// TwinCAT 3 PLC project Stage
// Title: Stage
// Company: _
// Author: Krystian Lis et al.
// ProjectVersion: 4.1.3
// ProgramVersion: 3.1.4026.22
// libraries:
//   Tc2_Standard, * (Beckhoff Automation GmbH)
//   Tc2_System, * (Beckhoff Automation GmbH)
//   Tc2_Utilities, * (Beckhoff Automation GmbH)
// project tree:
//   Plant/Debugging/ DebugStruct.TcDUT, I_Debug.TcIO
//   Plant/Entity/ Entity.TcPOU, I_Entity.TcIO, _I_Entity.TcIO
//   Plant/Execute/ Execute.TcPOU, I_Execute.TcIO, _I_Execute.TcIO
//   Plant/Init/ I_Init.TcIO
//   Plant/Job/ I_Worker.TcIO, _I_Worker.TcIO, Worker.TcPOU, I_Job.TcIO, JobState.TcDUT
//   Plant/OnlineChange/ I_OnlineChange.TcIO
//   Plant/ Plant.TcPOU, _Plant.TcGVL
//   Plant/PreInit/ I_PreInit.TcIO
//   Plant/PostInit/ I_PostInit.TcIO
//   Plant/Thread/ I_Thread.TcIO, Thread.TcPOU, _I_Thread.TcIO
//   Plant/Validate/ _I_ValidateGeneric.TcIO, I_ValidateInterface.TcIO
//   Utils/Color/ Argb.TcDUT, Argbb.TcPOU, GenArgb.TcPOU
//   Utils/Generic/ I_Generic.TcIO
//   Utils/Math/ Math.TcPOU
//   Utils/Path/ I_Path.TcIO, Path.TcPOU
//   Utils/Result/Error/ GenericResult.TcGVL
//   Utils/Result/ IsErr.TcPOU, IsFail.TcPOU, IsNone.TcPOU, IsOk.TcPOU, IsSome.TcPOU, Result.TcDUT
//   Utils/Strings/Alias/ Ch.TcDUT, Str.TcDUT
//   Utils/Strings/Strb/ I_Strb.TcIO, Strb.TcPOU
//   Utils/Strings/Strf/ Strf.TcPOU
//   Utils/Time/ GetTaskCycleTime.TcPOU, GetUnixTime.TcPOU
//   _/ Param.TcGVL
// real-time tasks:
//   TASK Example: cycle T#10ms, priority 20, ADS port 350
//   TASK Test: cycle T#10ms, priority 21, ADS port 351
//   TASK VISU_TASK: cycle T#200000us, priority 30, ADS port 352
//   TASK PlcTask: cycle T#10ms, priority 22, ADS port 353
//   TASK PlcTask1: cycle T#10ms, priority 23, ADS port 354
//   TASK PlcTask2: cycle T#10ms, priority 24, ADS port 355

// ---- Plant/Debugging/DebugStruct.TcDUT
// One diagnostic entry.
TYPE DebugStruct :
STRUCT
	iSource: I_Debug; // Object that reported the message.
	sComment: Str; // Diagnostic text.
END_STRUCT
END_TYPE

// ---- Plant/Job/JobState.TcDUT
// Worker lifecycle state.
{attribute 'qualified_only'}
{attribute 'strict'}
{attribute 'to_string'}
TYPE JobState :
(
	Idle, // Not attached to a thread.
	Init, // Will call JobInit next.
	Busy, // Calls JobExecute each worker cycle.
	Done // Will call JobExit and detach.
	
) BYTE;
END_TYPE

// ---- Utils/Color/Argb.TcDUT
// Packed ARGB color value.
TYPE Argb : DWORD; END_TYPE

// ---- Utils/Result/Result.TcDUT
// Result code: >0 Ok, 0 None, <0 Error.
TYPE Result : INT; END_TYPE

// ---- Utils/Strings/Alias/Ch.TcDUT
// Single-character string alias.
TYPE Ch : STRING(1); END_TYPE

// ---- Utils/Strings/Alias/Str.TcDUT
// Common 255-character string alias.
TYPE Str : STRING(255); END_TYPE

// ---- Plant/_Plant.TcGVL
{attribute 'qualified_only'}
{attribute 'global_init_slot' := '40001'}
VAR_GLOBAL INTERNAL
	panic: ARRAY[1..PARAM.MAX_PANIC_MSG] OF DebugStruct;
	warn: ARRAY[1..PARAM.MAX_WARN_MSG] OF DebugStruct;
	
	nLastPanic: UDINT := 1;
	nLastWarn: UDINT := 1;
	nTotalPanic: UDINT;
	nTotalWarn: UDINT;
	
	{attribute 'init_on_onlchange'}
	bOnlineChange: BOOL := TRUE;
	
	{attribute 'no_copy'}
	{attribute 'no_init'}
	bOnlineChangeEntityCreated: BOOL := FALSE;
	{attribute 'no_copy'}
	{attribute 'no_init'}
	bOnlineChangeEntityDeleted: BOOL := FALSE;

	iFirstThread: I_Thread;
	iLastThread: I_Thread;

	iFirstWorker: I_Worker;
	iLastWorker: I_Worker;
	
	MainThread: Thread;
	
	iFirstEntity: I_Entity;
	iLastEntity: I_Entity;
	
	bPanic: BOOL;
	bInit: BOOL := TRUE;
END_VAR

// ---- Utils/Result/Error/GenericResult.TcGVL
VAR_GLOBAL CONSTANT
	None	: Result := 0; // No result or end of iteration.
	Ok		: Result := 1; // Generic success.
	Error	: Result := -1; // Generic error.
END_VAR

// ---- _/Param.TcGVL
// Stage diagnostic buffer limits.
{attribute 'qualified_only'}
VAR_GLOBAL CONSTANT
	MAX_PANIC_MSG: UDINT(1..16#7FFFFFFF) := 10; // Panic buffer entries; do not set to 0.
	MAX_WARN_MSG: UDINT(1..16#7FFFFFFF) := 10; // Warning buffer entries; do not set to 0.
	VALIDATION_GUARD: UDINT(1..16#7FFFFFFF) := 100_000;
END_VAR

// ---- Plant/Debugging/I_Debug.TcIO
// Diagnostic marker interface.
INTERFACE I_Debug

END_INTERFACE

// ---- Plant/Entity/I_Entity.TcIO
// Registered entity handle.
INTERFACE I_Entity EXTENDS _I_Entity

// Raw discoverable interface for __QUERYINTERFACE.
PROPERTY Raw : I_Generic
GET
END_GET
END_PROPERTY

END_INTERFACE

// ---- Plant/Entity/_I_Entity.TcIO
INTERFACE INTERNAL _I_Entity EXTENDS I_Debug, I_ValidateInterface

METHOD INTERNAL GetNext : I_Entity
END_METHOD

METHOD INTERNAL SetNext
VAR_INPUT
	iNext: I_Entity;
END_VAR
END_METHOD

METHOD INTERNAL GetPrev : I_Entity
END_METHOD

METHOD INTERNAL SetPrev
VAR_INPUT
	iPrev: I_Entity;
END_VAR
END_METHOD

METHOD INTERNAL GetRaw : I_Generic
END_METHOD

METHOD INTERNAL SetRaw
VAR_INPUT
	iRaw: I_Generic;
END_VAR
END_METHOD

PROPERTY INTERNAL _Result : Result
GET
END_GET
END_PROPERTY

PROPERTY INTERNAL _NewInstance : BOOL
GET
END_GET
SET
END_SET
END_PROPERTY

END_INTERFACE

// ---- Plant/Execute/I_Execute.TcIO
// Cyclic callback contract; Execute is called once per assigned thread cycle.
INTERFACE I_Execute EXTENDS I_Debug

// Called cyclically by the assigned Stage thread.
METHOD Execute
END_METHOD

END_INTERFACE

// ---- Plant/Execute/_I_Execute.TcIO
INTERFACE INTERNAL _I_Execute EXTENDS I_Debug, I_ValidateInterface;

METHOD INTERNAL _Exe
VAR_OUTPUT
	iNext: _I_Execute;
END_VAR
END_METHOD

METHOD INTERNAL GetNext : _I_Execute
END_METHOD

METHOD INTERNAL SetNext
VAR_INPUT
	iNext: _I_Execute;
END_VAR
END_METHOD

METHOD INTERNAL GetPrev : _I_Execute
END_METHOD

METHOD INTERNAL SetPrev
VAR_INPUT
	iPrev: _I_Execute;
END_VAR
END_METHOD

METHOD INTERNAL GetThread : I_Thread
END_METHOD

METHOD INTERNAL SetThread
VAR_INPUT
	iThread: I_Thread;
END_VAR
END_METHOD

END_INTERFACE

// ---- Plant/Init/I_Init.TcIO
// Startup hook called after PreInit and before PostInit.
INTERFACE I_Init EXTENDS I_Generic

// Called once during Plant startup.
METHOD Init
END_METHOD

END_INTERFACE

// ---- Plant/Job/I_Worker.TcIO
// Public command interface for a Worker.
INTERFACE I_Worker EXTENDS _I_Worker

// Starts idle job; returns Ok attached, None command busy, Error invalid state or job.
METHOD Start : Result
VAR_INPUT
END_VAR
END_METHOD

// Current worker state.
PROPERTY State : JobState
GET
END_GET
END_PROPERTY

// Requests stop; Busy moves to Done and calls JobExit before returning Idle.
METHOD Stop
VAR_INPUT
END_VAR
END_METHOD

END_INTERFACE

// ---- Plant/Job/_I_Worker.TcIO
INTERFACE INTERNAL _I_Worker EXTENDS I_Debug, I_ValidateInterface;

METHOD INTERNAL GetNext : I_Worker
END_METHOD

METHOD INTERNAL SetNext
VAR_INPUT
	iNext: I_Worker;
END_VAR
END_METHOD

METHOD INTERNAL GetPrev : I_Worker
END_METHOD

METHOD INTERNAL SetPrev
VAR_INPUT
	iPrev: I_Worker;
END_VAR
END_METHOD

METHOD INTERNAL GetPlantNext : I_Worker
END_METHOD

METHOD INTERNAL SetPlantNext
VAR_INPUT
	iNext: I_Worker;
END_VAR
END_METHOD

METHOD INTERNAL GetPlantPrev : I_Worker
END_METHOD

METHOD INTERNAL SetPlantPrev
VAR_INPUT
	iPrev: I_Worker;
END_VAR
END_METHOD

METHOD INTERNAL Process
VAR_OUTPUT
	iNext: I_Worker;
END_VAR
END_METHOD

METHOD INTERNAL GetThread : I_Thread
END_METHOD

METHOD INTERNAL SetThread
VAR_INPUT
	iThread: I_Thread;
END_VAR
END_METHOD

END_INTERFACE

// ---- Plant/Job/I_Job.TcIO
// Startable job contract processed by Worker.
INTERFACE I_Job EXTENDS I_Debug

// Called every worker cycle while Busy.
METHOD JobExecute
VAR_INPUT
END_VAR
END_METHOD

// Called once when the worker leaves Done.
METHOD JobExit
VAR_INPUT
END_VAR
END_METHOD

// Called once when the worker enters Init.
METHOD JobInit
VAR_INPUT
END_VAR
END_METHOD

END_INTERFACE

// ---- Plant/OnlineChange/I_OnlineChange.TcIO
INTERFACE I_OnlineChange EXTENDS I_Generic

METHOD OnOnlineChange
VAR_INPUT
	bEntityDeleted: BOOL;
	bEntityCreated: BOOL;
END_VAR
END_METHOD

END_INTERFACE

// ---- Plant/PreInit/I_PreInit.TcIO
// Startup hook called before Init and PostInit.
INTERFACE I_PreInit EXTENDS I_Generic

// Called once during Plant startup before Init.
METHOD PreInit
END_METHOD

END_INTERFACE

// ---- Plant/PostInit/I_PostInit.TcIO
// Startup hook called after PreInit and Init.
INTERFACE I_PostInit EXTENDS I_Generic

// Called once during Plant startup after Init.
METHOD PostInit
END_METHOD

END_INTERFACE

// ---- Plant/Thread/I_Thread.TcIO
// Identifies a Stage execution thread.
INTERFACE I_Thread EXTENDS _I_Thread

END_INTERFACE

// ---- Plant/Thread/_I_Thread.TcIO
INTERFACE INTERNAL _I_Thread EXTENDS I_Debug, I_ValidateInterface

METHOD INTERNAL GetFirst : _I_Execute
END_METHOD

METHOD INTERNAL GetFirstWorker : I_Worker
END_METHOD

METHOD INTERNAL GetLast : _I_Execute
END_METHOD

METHOD INTERNAL GetLastWorker : I_Worker
END_METHOD

METHOD INTERNAL GetNext : I_Thread
END_METHOD

METHOD INTERNAL SetNext
VAR_INPUT
	iNext: I_Thread;
END_VAR
END_METHOD

METHOD INTERNAL GetPrev : I_Thread
END_METHOD

METHOD INTERNAL SetPrev
VAR_INPUT
	iPrev: I_Thread;
END_VAR
END_METHOD

METHOD INTERNAL AttachExecute : Result
VAR_INPUT
	iExecute: _I_Execute;
END_VAR
END_METHOD

METHOD INTERNAL AttachWorker : Result
VAR_INPUT
	iWorker: I_Worker;
END_VAR
END_METHOD

METHOD INTERNAL DetachExecute : Result
VAR_INPUT
	iExecute: _I_Execute;
END_VAR
END_METHOD

METHOD INTERNAL DetachWorker : Result
VAR_INPUT
	iWorker: I_Worker;
END_VAR
END_METHOD

METHOD INTERNAL ValidateThread : Result
END_METHOD

END_INTERFACE

// ---- Plant/Validate/_I_ValidateGeneric.TcIO
INTERFACE INTERNAL _I_ValidateGeneric EXTENDS __SYSTEM.IQueryInterface, I_Debug

END_INTERFACE

// ---- Plant/Validate/I_ValidateInterface.TcIO
INTERFACE I_ValidateInterface EXTENDS I_Debug

{attribute 'hide'}
METHOD ValidateInterface
VAR_INPUT
END_VAR
END_METHOD

END_INTERFACE

// ---- Utils/Generic/I_Generic.TcIO
// Common discoverable base interface for registered entities.
INTERFACE I_Generic EXTENDS __SYSTEM.IQueryInterface, I_Debug

END_INTERFACE

// ---- Utils/Path/I_Path.TcIO
// Path identifier interface.
INTERFACE I_Path

// Full generated path including options.
PROPERTY Get : Str
GET
END_GET
END_PROPERTY

// TRUE when the path contains sSegment.
METHOD Has : BOOL
VAR_INPUT
	sSegment: Str; // Segment to find.
END_VAR
END_METHOD

// Full path length including options.
PROPERTY Length : USINT
GET
END_GET
END_PROPERTY

// Generated path without options.
PROPERTY Name : Str
GET
END_GET
END_PROPERTY

// Optional query-style path segment.
PROPERTY Option : Str
GET
END_GET
SET
END_SET
END_PROPERTY

END_INTERFACE

// ---- Utils/Strings/Strb/I_Strb.TcIO
// Chainable string builder interface.
INTERFACE INTERNAL I_Strb EXTENDS I_Debug

// Appends text; truncates at 255 chars.
METHOD Append : I_Strb
VAR_INPUT
    sToAdd : Str; // Text to append.
END_VAR
END_METHOD

// Finds first match after position; outputs zero positions when not found.
METHOD FindFirstAfter : I_Strb
VAR_INPUT
    sToFind : Str;      // Text to find.
    nPosition : INT := 1; // One-based start position.
END_VAR
VAR_OUTPUT
    nStart : INT;       // Match start, or 0.
    nEnd : INT;         // Match end, or 0.
END_VAR
END_METHOD

// Finds last match before position; outputs zero positions when not found.
METHOD FindLastBefore : I_Strb
VAR_INPUT
    sToFind : Str;        // Text to find.
    nPosition : INT := 256; // One-based end position; 256 means current length.
END_VAR
VAR_OUTPUT
    nStart : INT;         // Match start, or 0.
    nEnd : INT;           // Match end, or 0.
END_VAR
END_METHOD

// Returns current text.
METHOD Get : Str
VAR_INPUT
END_VAR
END_METHOD

// Returns current length.
METHOD GetLength : INT
VAR_INPUT
END_VAR
END_METHOD

// TRUE when text is found after position.
METHOD HasAfter : BOOL
VAR_INPUT
    sToFind : Str;      // Text to find.
    nPosition : INT := 0; // One-based start position.
END_VAR
VAR_OUTPUT
    nStart : INT;       // Match start, or 0.
    nEnd : INT;         // Match end, or 0.
END_VAR
END_METHOD

// TRUE when text is found before position.
METHOD HasBefore : BOOL
VAR_INPUT
    sToFind : Str;        // Text to find.
    nPosition : INT := 256; // One-based end position; 256 means current length.
END_VAR
VAR_OUTPUT
    nStart : INT;         // Match start, or 0.
    nEnd : INT;           // Match end, or 0.
END_VAR
END_METHOD

// Inserts text; no change when position is invalid.
METHOD Inject : I_Strb
VAR_INPUT
    nPosition : INT;    // One-based insert position.
    sToInject : Str;    // Text to insert.
END_VAR
END_METHOD

// TRUE when current length is 0.
METHOD IsEmpty : BOOL
VAR_INPUT
END_VAR
END_METHOD

// Outputs current length and returns this builder.
METHOD Length : I_Strb
VAR_OUTPUT
	nLen: INT; // Current length.
END_VAR
END_METHOD

// Prepends text; truncates at 255 chars.
METHOD Prepend : I_Strb
VAR_INPUT
    sToAdd : Str; // Text to prepend.
END_VAR
END_METHOD

// Removes text; no change when position or length is invalid.
METHOD Remove : I_Strb
VAR_INPUT
    nLength : INT;    // Characters to remove.
    nPosition : INT;  // One-based start position.
END_VAR
END_METHOD

// Sets current text.
METHOD Set : I_Strb
VAR_INPUT
    sValue : Str; // New text.
END_VAR
END_METHOD

// Copies substring into sSlice; no change when position or length is invalid.
METHOD Slice : I_Strb
VAR_INPUT
	nLength : INT;   // Characters to copy.
    nPosition : INT; // One-based start position.
END_VAR
VAR_OUTPUT
    sSlice : Strb;   // Output slice builder.
END_VAR
END_METHOD

// Splits text into left and right builders.
METHOD Split : I_Strb
VAR_INPUT
    nPosition : INT; // One-based split position.
END_VAR
VAR_OUTPUT
    sLeft : Strb;    // Left side.
    sRight : Strb;   // Right side.
END_VAR
END_METHOD

// Outputs current text and returns this builder.
METHOD Write : I_Strb;
VAR_OUTPUT
	sOut: Str; // Current text.
END_VAR
END_METHOD

END_INTERFACE

// ---- Plant/Thread/Thread.TcPOU
// Runs executors and active workers assigned to this TwinCAT task.
FUNCTION_BLOCK Thread IMPLEMENTS I_Thread
VAR
	iFirstExecute: _I_Execute;
	iLastExecute: _I_Execute;

	iFirstWorker: I_Worker;
	iLastWorker: I_Worker;

	iPrevThread: I_Thread;
	iNextThread: I_Thread;
END_VAR

METHOD INTERNAL AttachExecute : Result
VAR_INPUT
	iExecute: _I_Execute;
END_VAR
VAR
	iThis: I_Thread := THIS^;
	iThread: I_Thread;
	iPrev: _I_Execute;
	iNext: _I_Execute;
END_VAR
IF iExecute = 0 THEN
	AttachExecute := Error;
	RETURN;
END_IF

iThread := iExecute.GetThread();
IF iThread <> iThis THEN
	AttachExecute := Error;
	RETURN;
END_IF

iPrev := iExecute.GetPrev();
iNext := iExecute.GetNext();

IF iPrev <> 0 OR iNext <> 0 OR
	iFirstExecute = iExecute OR iLastExecute = iExecute THEN
	Plant.Warn(iExecute, 'Execute attach skipped: execute is already linked in a thread execute list.');
	AttachExecute := None;
    RETURN;
END_IF

iExecute.SetPrev(iLastExecute);
iExecute.SetNext(0);

IF iLastExecute <> 0 THEN
	iLastExecute.SetNext(iExecute);
	iLastExecute := iExecute;
ELSE
	iFirstExecute := iExecute;
	iLastExecute  := iExecute;
END_IF

AttachExecute := Ok;
END_METHOD

METHOD INTERNAL AttachWorker : Result
VAR_INPUT
	iWorker: I_Worker;
END_VAR
VAR
	iThis: I_Thread := THIS^;
	iThread: I_Thread;
	iPrev: I_Worker;
	iNext: I_Worker;
END_VAR
IF iWorker = 0 THEN
	AttachWorker := Error;
	RETURN;
END_IF

iThread := iWorker.GetThread();
IF iThread <> iThis THEN
	AttachWorker := Error;
	RETURN;
END_IF

iPrev := iWorker.GetPrev();
iNext := iWorker.GetNext();

IF iPrev <> 0 OR iNext <> 0 OR
	iFirstWorker = iWorker OR iLastWorker = iWorker THEN
	Plant.Warn(iWorker, 'Worker attach skipped: worker is already linked in a thread worker list.');
	AttachWorker := None;
    RETURN;
END_IF

iWorker.SetPrev(iLastWorker);
iWorker.SetNext(0);

IF iLastWorker <> 0 THEN
	iLastWorker.SetNext(iWorker);
	iLastWorker := iWorker;
ELSE
	iFirstWorker := iWorker;
	iLastWorker  := iWorker;
END_IF

AttachWorker := Ok;
END_METHOD

METHOD INTERNAL DetachExecute : Result
VAR_INPUT
	iExecute: _I_Execute;
END_VAR
VAR
	iThis: I_Thread := THIS^;
	iThread: I_Thread;
	iPrev : _I_Execute;
	iNext : _I_Execute;
END_VAR
IF iExecute = 0 THEN
	DetachExecute := Error;
	RETURN;
END_IF

iThread := iExecute.GetThread();
IF iThread <> iThis THEN
	DetachExecute := Error;
	RETURN;
END_IF

iPrev := iExecute.GetPrev();
iNext := iExecute.GetNext();

IF iPrev <> 0 THEN
    iPrev.SetNext(iNext);
END_IF

IF iNext <> 0 THEN
    iNext.SetPrev(iPrev);
END_IF

IF iFirstExecute = iExecute THEN
    iFirstExecute := iNext;
END_IF

IF iLastExecute = iExecute THEN
    iLastExecute := iPrev;
END_IF

iExecute.SetPrev(0);
iExecute.SetNext(0);

DetachExecute := Ok;
END_METHOD

METHOD INTERNAL DetachWorker : Result
VAR_INPUT
	iWorker: I_Worker;
END_VAR
VAR
	iThis: I_Thread := THIS^;
	iThread: I_Thread;
	iNext: I_Worker;
	iPrev: I_Worker;
END_VAR
IF iWorker = 0 THEN
	DetachWorker := Error;
	RETURN;
END_IF

iThread := iWorker.GetThread();
IF iThread <> iThis THEN
	DetachWorker := Error;
	RETURN;
END_IF

iPrev := iWorker.GetPrev();
iNext := iWorker.GetNext();

IF iPrev <> 0 THEN
    iPrev.SetNext(iNext);
END_IF

IF iNext <> 0 THEN
    iNext.SetPrev(iPrev);
END_IF

IF iFirstWorker = iWorker THEN
    iFirstWorker := iNext;
END_IF

IF iLastWorker = iWorker THEN
    iLastWorker := iPrev;
END_IF

iWorker.SetPrev(0);
iWorker.SetNext(0);

DetachWorker := Ok;
END_METHOD

{attribute 'hide'}
METHOD FB_Exit : BOOL
VAR_INPUT
	bInCopyCode: BOOL;
END_VAR
VAR
	iThis: I_Thread := THIS^;
	iMainThread: I_Thread := _Plant.MainThread;
	iExecute: _I_Execute;
	iWorker: I_Worker;
END_VAR
IF NOT bInCopyCode THEN
	IF iThis <> iMainThread THEN
		WHILE iFirstExecute <> 0 DO
			iExecute := iFirstExecute;
			iExecute.SetThread(iThis);

			IF DetachExecute(iExecute) <> Ok THEN
				Plant.Panic(iExecute, 'Thread exit failed: could not detach execute before moving it to MainThread.');
				EXIT;
			END_IF

			iExecute.SetThread(iMainThread);

			IF IsErr(iMainThread.AttachExecute(iExecute)) THEN
				Plant.Panic(iExecute, 'Thread exit failed: could not attach execute to MainThread before detaching thread.');
				EXIT;
			END_IF

			Plant.Warn(iExecute, 'Thread exit transfer: owning thread left scope; moved execute to MainThread.');
		END_WHILE

		WHILE iFirstWorker <> 0 DO
			iWorker := iFirstWorker;
			iWorker.SetThread(iThis);

			IF DetachWorker(iWorker) <> Ok THEN
				Plant.Panic(iWorker, 'Thread exit failed: could not detach worker before moving it to MainThread.');
				EXIT;
			END_IF

			iWorker.SetThread(iMainThread);

			IF IsErr(iMainThread.AttachWorker(iWorker)) THEN
				Plant.Panic(iWorker, 'Thread exit failed: could not attach worker to MainThread before detaching thread.');
				EXIT;
			END_IF

			Plant.Warn(iWorker, 'Thread exit transfer: owning thread left scope; moved worker to MainThread.');
		END_WHILE
	END_IF

	Plant._DetachThread(THIS^);
END_IF
END_METHOD

{attribute 'hide'}
METHOD FB_Init : BOOL
VAR_INPUT
	bInitRetains: BOOL;
	bInCopyCode: BOOL;
END_VAR
IF bInCopyCode THEN
	RETURN;
END_IF

IF IsErr(Plant._AttachThread(THIS^)) THEN
	Plant.Panic(THIS^, 'Thread initialization failed: could not attach thread to Plant registry.');
END_IF
END_METHOD

METHOD INTERNAL GetFirst : _I_Execute
GetFirst := iFirstExecute;
END_METHOD

METHOD INTERNAL GetFirstWorker : I_Worker
GetFirstWorker := iFirstWorker;
END_METHOD

METHOD INTERNAL GetLast : _I_Execute
GetLast := iLastExecute;
END_METHOD

METHOD INTERNAL GetLastWorker : I_Worker
GetLastWorker := iLastWorker;
END_METHOD

METHOD INTERNAL GetNext : I_Thread
GetNext := iNextThread;
END_METHOD

METHOD INTERNAL GetPrev : I_Thread
GetPrev := iPrevThread;
END_METHOD

// Processes active workers, then cyclic executors; returns during init or panic.
METHOD Run
VAR
	iWorker: I_Worker := iFirstWorker;
	iExecute: _I_Execute := iFirstExecute;
END_VAR
IF Plant.IsInit OR Plant.Panicked THEN
	RETURN;
END_IF

WHILE iWorker <> 0 DO
	iWorker.Process(iNext => iWorker);
END_WHILE

WHILE iExecute <> 0 DO
	iExecute._Exe(iNext => iExecute);
END_WHILE
END_METHOD

METHOD INTERNAL SetNext
VAR_INPUT
	iNext: I_Thread;
END_VAR
iNextThread := iNext;
END_METHOD

METHOD INTERNAL SetPrev
VAR_INPUT
	iPrev: I_Thread;
END_VAR
iPrevThread := iPrev;
END_METHOD

{attribute 'hide'}
METHOD ValidateInterface
VAR_INPUT
END_VAR
END_METHOD

METHOD INTERNAL ValidateThread : Result
VAR CONSTANT
	GUARD: UDINT := Param.VALIDATION_GUARD;
END_VAR
VAR
	iThis: I_Thread := THIS^;
	iExecute: _I_Execute;
	iPrevExecute: _I_Execute;
	iNextExecute: _I_Execute;
	iExecuteThread: I_Thread;
	iWorker: I_Worker;
	iPrevWorker: I_Worker;
	iNextWorker: I_Worker;
	iWorkerThread: I_Thread;
	iCheckExecute: _I_Execute;
	iCheckWorker: I_Worker;
	nGuard: UDINT;
	_err: __SYSTEM.ExceptionCode;
END_VAR
ValidateThread := Error;

__TRY
	IF iFirstExecute = 0 THEN
		IF iLastExecute <> 0 THEN
			Plant.Panic(THIS^, 'Thread validation failed: first execute is 0 but last execute is not 0.');
			RETURN;
		END_IF
	ELSE
		IF Plant.ValidateInterface(iFirstExecute) <> Ok THEN
			Plant.Panic(THIS^, 'Thread validation failed: first execute did not pass ValidateInterface.');
			RETURN;
		END_IF

		IF iLastExecute = 0 THEN
			Plant.Panic(THIS^, 'Thread validation failed: first execute is not 0 but last execute is 0.');
			RETURN;
		END_IF

		IF Plant.ValidateInterface(iLastExecute) <> Ok THEN
			Plant.Panic(THIS^, 'Thread validation failed: last execute did not pass ValidateInterface.');
			RETURN;
		END_IF

		iCheckExecute := iFirstExecute.GetPrev();
		IF iCheckExecute <> 0 THEN
			Plant.Panic(iFirstExecute, 'Thread validation failed: first execute has a nonzero _Prev link.');
			RETURN;
		END_IF

		iCheckExecute := iLastExecute.GetNext();
		IF iCheckExecute <> 0 THEN
			Plant.Panic(iLastExecute, 'Thread validation failed: last execute has a nonzero _Next link.');
			RETURN;
		END_IF
	END_IF

	iExecute := iFirstExecute;
	iPrevExecute := 0;
	nGuard := 0;

	WHILE iExecute <> 0 DO
		nGuard := nGuard + 1;
		IF nGuard > GUARD THEN
			Plant.Panic(THIS^, 'Thread validation failed: execute traversal exceeded GUARD; probable cycle.');
			RETURN;
		END_IF

		IF Plant.ValidateInterface(iExecute) <> Ok THEN
			Plant.Panic(THIS^, 'Thread validation failed: current execute did not pass ValidateInterface before link access.');
			RETURN;
		END_IF

		iCheckExecute := iExecute.GetPrev();
		IF iCheckExecute <> iPrevExecute THEN
			Plant.Panic(iExecute, 'Thread validation failed: current execute _Prev does not match previous visited execute.');
			RETURN;
		END_IF

		iExecuteThread := iExecute.GetThread();
		IF Plant.ValidateInterface(iExecuteThread) <> Ok THEN
			Plant.Panic(iExecute, 'Thread validation failed: current execute _Thread is 0 or failed ValidateInterface.');
			RETURN;
		END_IF

		IF iExecuteThread <> iThis THEN
			Plant.Panic(iExecute, 'Thread validation failed: current execute _Thread does not point to the owning thread.');
			RETURN;
		END_IF

		iNextExecute := iExecute.GetNext();

		IF iNextExecute <> 0 THEN
			IF Plant.ValidateInterface(iNextExecute) <> Ok THEN
				Plant.Panic(iExecute, 'Thread validation failed: current execute _Next did not pass ValidateInterface.');
				RETURN;
			END_IF

			IF iNextExecute = iExecute THEN
				Plant.Panic(iExecute, 'Thread validation failed: current execute _Next points to itself.');
				RETURN;
			END_IF

			iCheckExecute := iNextExecute.GetPrev();
			IF iCheckExecute <> iExecute THEN
				Plant.Panic(iExecute, 'Thread validation failed: next execute _Prev does not point back to current execute.');
				RETURN;
			END_IF
		END_IF

		iPrevExecute := iExecute;
		iExecute := iNextExecute;
	END_WHILE

	IF iPrevExecute <> iLastExecute THEN
		Plant.Panic(THIS^, 'Thread validation failed: last visited execute does not match thread last execute.');
		RETURN;
	END_IF

	IF iFirstWorker = 0 THEN
		IF iLastWorker <> 0 THEN
			Plant.Panic(THIS^, 'Thread validation failed: first worker is 0 but last worker is not 0.');
			RETURN;
		END_IF
	ELSE
		IF Plant.ValidateInterface(iFirstWorker) <> Ok THEN
			Plant.Panic(THIS^, 'Thread validation failed: first worker did not pass ValidateInterface.');
			RETURN;
		END_IF

		IF iLastWorker = 0 THEN
			Plant.Panic(THIS^, 'Thread validation failed: first worker is not 0 but last worker is 0.');
			RETURN;
		END_IF

		IF Plant.ValidateInterface(iLastWorker) <> Ok THEN
			Plant.Panic(THIS^, 'Thread validation failed: last worker did not pass ValidateInterface.');
			RETURN;
		END_IF

		iCheckWorker := iFirstWorker.GetPrev();
		IF iCheckWorker <> 0 THEN
			Plant.Panic(iFirstWorker, 'Thread validation failed: first worker has a nonzero _Prev link.');
			RETURN;
		END_IF

		iCheckWorker := iLastWorker.GetNext();
		IF iCheckWorker <> 0 THEN
			Plant.Panic(iLastWorker, 'Thread validation failed: last worker has a nonzero _Next link.');
			RETURN;
		END_IF
	END_IF

	iWorker := iFirstWorker;
	iPrevWorker := 0;
	nGuard := 0;

	WHILE iWorker <> 0 DO
		nGuard := nGuard + 1;
		IF nGuard > GUARD THEN
			Plant.Panic(THIS^, 'Thread validation failed: worker traversal exceeded GUARD; probable cycle.');
			RETURN;
		END_IF

		IF Plant.ValidateInterface(iWorker) <> Ok THEN
			Plant.Panic(THIS^, 'Thread validation failed: current worker did not pass ValidateInterface before link access.');
			RETURN;
		END_IF

		iCheckWorker := iWorker.GetPrev();
		IF iCheckWorker <> iPrevWorker THEN
			Plant.Panic(iWorker, 'Thread validation failed: current worker _Prev does not match previous visited worker.');
			RETURN;
		END_IF

		iWorkerThread := iWorker.GetThread();
		IF Plant.ValidateInterface(iWorkerThread) <> Ok THEN
			Plant.Panic(iWorker, 'Thread validation failed: current worker Thread is 0 or failed ValidateInterface.');
			RETURN;
		END_IF

		IF iWorkerThread <> iThis THEN
			Plant.Panic(iWorker, 'Thread validation failed: current worker Thread does not point to the owning thread.');
			RETURN;
		END_IF

		iNextWorker := iWorker.GetNext();

		IF iNextWorker <> 0 THEN
			IF Plant.ValidateInterface(iNextWorker) <> Ok THEN
				Plant.Panic(iWorker, 'Thread validation failed: current worker _Next did not pass ValidateInterface.');
				RETURN;
			END_IF

			IF iNextWorker = iWorker THEN
				Plant.Panic(iWorker, 'Thread validation failed: current worker _Next points to itself.');
				RETURN;
			END_IF

			iCheckWorker := iNextWorker.GetPrev();
			IF iCheckWorker <> iWorker THEN
				Plant.Panic(iWorker, 'Thread validation failed: next worker _Prev does not point back to current worker.');
				RETURN;
			END_IF
		END_IF

		iPrevWorker := iWorker;
		iWorker := iNextWorker;
	END_WHILE

	IF iPrevWorker <> iLastWorker THEN
		Plant.Panic(THIS^, 'Thread validation failed: last visited worker does not match thread last worker.');
		RETURN;
	END_IF

	ValidateThread := Ok;

__CATCH(_err)
	Plant.Panic(THIS^, 'Thread validation failed: exception while reading validation interfaces or links.');
	ValidateThread := Error;
__ENDTRY
END_METHOD

END_FUNCTION_BLOCK

// ---- Plant/Plant.TcPOU
// Stage runtime: startup hooks, entity registry, main-thread execution, and diagnostics.
PROGRAM Plant

METHOD INTERNAL _AttachEntity : Result
VAR_INPUT
	iEntity: I_Entity;
END_VAR
IF iEntity = 0 THEN
	Plant.Panic(0, 'Entity = 0!');
	_AttachEntity := Error;

ELSIF IsSome(iEntity._Result) THEN
	Plant.Warn(iEntity, 'Entity attach skipped: entity is already attached to the Plant entity registry.');
	_AttachEntity := None;
	RETURN;

ELSIF _Plant.iLastEntity <> 0 AND _Plant.iFirstEntity <> 0 THEN
	_Plant.iLastEntity.SetNext(iEntity);
	iEntity.SetPrev(_Plant.iLastEntity);
	_Plant.iLastEntity := iEntity;
	_AttachEntity := Ok;

ELSIF _Plant.iLastEntity = 0 AND _Plant.iFirstEntity = 0 THEN
	_Plant.iFirstEntity := iEntity;
	_Plant.iLastEntity := iEntity;
	_AttachEntity := Ok;

ELSE
	_AttachEntity := Error;

END_IF
END_METHOD

METHOD INTERNAL _AttachThread : Result
VAR_INPUT
	iThread: I_Thread;
END_VAR
VAR
	iPrev: I_Thread;
	iNext: I_Thread;
END_VAR
IF iThread = 0 THEN
	Plant.Panic(0, 'Thread attach failed: thread is 0.');
	_AttachThread := Error;
	RETURN;
END_IF

iPrev := iThread.GetPrev();
iNext := iThread.GetNext();

IF iPrev <> 0 OR iNext <> 0 OR
	_Plant.iFirstThread = iThread OR _Plant.iLastThread = iThread THEN
	Plant.Warn(iThread, 'Thread attach skipped: thread is already linked in the Plant thread registry.');
	_AttachThread := None;
	RETURN;
END_IF

iThread.SetPrev(_Plant.iLastThread);
iThread.SetNext(0);

IF _Plant.iLastThread <> 0 THEN
	_Plant.iLastThread.SetNext(iThread);
	_Plant.iLastThread := iThread;
ELSE
	_Plant.iFirstThread := iThread;
	_Plant.iLastThread := iThread;
END_IF

_AttachThread := Ok;
END_METHOD

METHOD INTERNAL _AttachWorker : Result
VAR_INPUT
	iWorker: I_Worker;
END_VAR
VAR
	iPlantPrev: I_Worker;
	iPlantNext: I_Worker;
END_VAR
IF iWorker = 0 THEN
	Plant.Panic(0, 'Worker attach failed: worker is 0.');
	_AttachWorker := Error;
	RETURN;
END_IF

iPlantPrev := iWorker.GetPlantPrev();
iPlantNext := iWorker.GetPlantNext();

IF iPlantPrev <> 0 OR iPlantNext <> 0 OR
	_Plant.iFirstWorker = iWorker OR _Plant.iLastWorker = iWorker THEN
	Plant.Warn(iWorker, 'Worker attach skipped: worker is already linked in the Plant worker registry.');
	_AttachWorker := None;
	RETURN;
END_IF

iWorker.SetPlantPrev(_Plant.iLastWorker);
iWorker.SetPlantNext(0);

IF _Plant.iLastWorker <> 0 THEN
	_Plant.iLastWorker.SetPlantNext(iWorker);
	_Plant.iLastWorker := iWorker;
ELSE
	_Plant.iFirstWorker := iWorker;
	_Plant.iLastWorker := iWorker;
END_IF

_AttachWorker := Ok;
END_METHOD

METHOD PRIVATE _CallInits
VAR
	_iInit: I_Init;
	_iEtt: I_Entity;
END_VAR
WHILE IsOk(Plant.NextEtt(_iEtt)) DO
	IF _iEtt._NewInstance THEN
		IF __QUERYINTERFACE(_iEtt.GetRaw(), _iInit) THEN
			_iInit.Init();
		END_IF
	END_IF
END_WHILE
END_METHOD

METHOD PRIVATE _CallOnlineChange
VAR
	_iOnlineChange: I_OnlineChange;
	_iEtt: I_Entity;
END_VAR
WHILE Plant.NextEtt(_iEtt) = Ok DO
	IF __QUERYINTERFACE(_iEtt.GetRaw(), _iOnlineChange) THEN
		_iOnlineChange.OnOnlineChange(
				bEntityDeleted := _Plant.bOnlineChangeEntityDeleted,
				bEntityCreated := _Plant.bOnlineChangeEntityCreated);
	END_IF
END_WHILE
END_METHOD

METHOD PRIVATE _CallPostInits
VAR
	_iPostInit: I_PostInit;
	_iEtt: I_Entity;
END_VAR
WHILE IsOk(Plant.NextEtt(_iEtt)) DO
	IF _iEtt._NewInstance THEN
		IF __QUERYINTERFACE(_iEtt.GetRaw(), _iPostInit) THEN
			_iPostInit.PostInit();
		END_IF
	END_IF
END_WHILE
END_METHOD

METHOD PRIVATE _CallPreInits
VAR
	_iPreInit: I_PreInit;
	_iEtt: I_Entity;
END_VAR
WHILE IsOk(Plant.NextEtt(_iEtt)) DO
	IF _iEtt._NewInstance THEN
		IF __QUERYINTERFACE(_iEtt.GetRaw(), _iPreInit) THEN
			_iPreInit.PreInit();
		END_IF
	END_IF
END_WHILE
END_METHOD

METHOD PRIVATE _ClearNewInstanceFlags
VAR
	_iEtt: I_Entity;
END_VAR
WHILE IsOk(Plant.NextEtt(_iEtt)) DO
	_iEtt._NewInstance := FALSE;
END_WHILE
END_METHOD

METHOD INTERNAL _DetachEntity : Result
VAR_INPUT
	iEntity: I_Entity;
END_VAR
VAR
	iPrev: I_Entity;
	iNext: I_Entity;
END_VAR
IF iEntity = 0 THEN
	_DetachEntity := Error;
	RETURN;
END_IF

iPrev := iEntity.GetPrev();
iNext := iEntity.GetNext();

IF iPrev = 0 AND iNext = 0 AND
	_Plant.iFirstEntity <> iEntity AND _Plant.iLastEntity <> iEntity THEN
	_DetachEntity := None;
	RETURN;
END_IF

IF iPrev <> 0 THEN
	iPrev.SetNext(iNext);
END_IF

IF iNext <> 0 THEN
	iNext.SetPrev(iPrev);
END_IF

IF _Plant.iFirstEntity = iEntity THEN
	_Plant.iFirstEntity := iNext;
END_IF

IF _Plant.iLastEntity = iEntity THEN
	_Plant.iLastEntity := iPrev;
END_IF

iEntity.SetPrev(0);
iEntity.SetNext(0);

_DetachEntity := Ok;
END_METHOD

METHOD INTERNAL _DetachThread : Result
VAR_INPUT
	iThread: I_Thread;
END_VAR
VAR
	iPrev: I_Thread;
	iNext: I_Thread;
END_VAR
IF iThread = 0 THEN
	_DetachThread := Error;
	RETURN;
END_IF

iPrev := iThread.GetPrev();
iNext := iThread.GetNext();

IF iPrev = 0
	AND iNext = 0
	AND _Plant.iFirstThread <> iThread
	AND _Plant.iLastThread <> iThread
THEN
	_DetachThread := None;
	RETURN;
END_IF

IF iPrev <> 0 THEN
	iPrev.SetNext(iNext);
END_IF

IF iNext <> 0 THEN
	iNext.SetPrev(iPrev);
END_IF

IF _Plant.iFirstThread = iThread THEN
	_Plant.iFirstThread := iNext;
END_IF

IF _Plant.iLastThread = iThread THEN
	_Plant.iLastThread := iPrev;
END_IF

iThread.SetPrev(0);
iThread.SetNext(0);

_DetachThread := Ok;
END_METHOD

METHOD INTERNAL _DetachWorker : Result
VAR_INPUT
	iWorker: I_Worker;
END_VAR
VAR
	iPrev: I_Worker;
	iNext: I_Worker;
END_VAR
IF iWorker = 0 THEN
	_DetachWorker := Error;
	RETURN;
END_IF

iPrev := iWorker.GetPlantPrev();
iNext := iWorker.GetPlantNext();

IF iPrev = 0 AND iNext = 0 AND
	_Plant.iFirstWorker <> iWorker AND _Plant.iLastWorker <> iWorker THEN
	_DetachWorker := None;
	RETURN;
END_IF

IF iPrev <> 0 THEN
	iPrev.SetPlantNext(iNext);
END_IF

IF iNext <> 0 THEN
	iNext.SetPlantPrev(iPrev);
END_IF

IF _Plant.iFirstWorker = iWorker THEN
	_Plant.iFirstWorker := iNext;
END_IF

IF _Plant.iLastWorker = iWorker THEN
	_Plant.iLastWorker := iPrev;
END_IF

iWorker.SetPlantPrev(0);
iWorker.SetPlantNext(0);

_DetachWorker := Ok;
END_METHOD

METHOD INTERNAL _IsThreadRegistered : BOOL
VAR_INPUT
	iThread: I_Thread;
END_VAR
VAR CONSTANT
	GUARD: UDINT := Param.VALIDATION_GUARD;
END_VAR
VAR
	iCurrent: I_Thread;
	nGuard: UDINT;
	_err: __SYSTEM.ExceptionCode;
END_VAR
_IsThreadRegistered := FALSE;

__TRY
	IF ValidateInterface(iThread) <> Ok THEN
		RETURN;
	END_IF

	iCurrent := _Plant.iFirstThread;

	WHILE iCurrent <> 0 DO
		nGuard := nGuard + 1;
		IF nGuard > GUARD THEN
			RETURN;
		END_IF

		IF ValidateInterface(iCurrent) <> Ok THEN
			RETURN;
		END_IF

		IF iCurrent = iThread THEN
			_IsThreadRegistered := TRUE;
			RETURN;
		END_IF

		iCurrent := iCurrent.GetNext();
	END_WHILE

__CATCH(_err)
	_IsThreadRegistered := FALSE;
__ENDTRY
END_METHOD

METHOD INTERNAL _ThreadDispatcher : Result
VAR_INPUT
	bWarn: BOOL;
END_VAR
VAR CONSTANT
	GUARD: UDINT := Param.VALIDATION_GUARD;
END_VAR
VAR
	iMainThread: I_Thread := _Plant.MainThread;
	iThread: I_Thread;
	iPrevThread: I_Thread;
	iNextThread: I_Thread;
	iExecute: _I_Execute;
	iPrevExecute: _I_Execute;
	iNextExecute: _I_Execute;
	iLastExecute: _I_Execute;
	iExecuteThread: I_Thread;
	iWorker: I_Worker;
	iPrevWorker: I_Worker;
	iNextWorker: I_Worker;
	iLastWorker: I_Worker;
	iWorkerThread: I_Thread;
	iCheckThread: I_Thread;
	iCheckExecute: _I_Execute;
	iCheckWorker: I_Worker;
	nThreadGuard: UDINT;
	nExecuteGuard: UDINT;
	nWorkerGuard: UDINT;
	bDefaultedThread: BOOL;
	bMoved: BOOL;
	_err: __SYSTEM.ExceptionCode;
END_VAR
_ThreadDispatcher := Error;

__TRY
	IF ValidateInterface(iMainThread) <> Ok THEN
		Plant.Panic(0, 'Thread dispatch failed: _Plant.MainThread is 0 or failed ValidateInterface.');
		RETURN;
	END_IF

	IF _Plant.iFirstThread = 0 THEN
		IF _Plant.iLastThread <> 0 THEN
			Plant.Panic(0, 'Thread dispatch failed: first thread is 0 but last thread is not 0.');
			RETURN;
		END_IF
	ELSE
		IF ValidateInterface(_Plant.iFirstThread) <> Ok THEN
			Plant.Panic(0, 'Thread dispatch failed: first thread failed ValidateInterface before list access.');
			RETURN;
		END_IF

		IF _Plant.iLastThread = 0 THEN
			Plant.Panic(0, 'Thread dispatch failed: first thread is not 0 but last thread is 0.');
			RETURN;
		END_IF

		IF ValidateInterface(_Plant.iLastThread) <> Ok THEN
			Plant.Panic(0, 'Thread dispatch failed: last thread failed ValidateInterface before list access.');
			RETURN;
		END_IF

		iCheckThread := _Plant.iFirstThread.GetPrev();
		IF iCheckThread <> 0 THEN
			Plant.Panic(_Plant.iFirstThread, 'Thread dispatch failed: first thread has a nonzero _Prev link.');
			RETURN;
		END_IF

		iCheckThread := _Plant.iLastThread.GetNext();
		IF iCheckThread <> 0 THEN
			Plant.Panic(_Plant.iLastThread, 'Thread dispatch failed: last thread has a nonzero _Next link.');
			RETURN;
		END_IF
	END_IF

	IF NOT Plant._IsThreadRegistered(iMainThread) THEN
		Plant.Panic(0, 'Thread dispatch failed: _Plant.MainThread is not linked in the Plant thread registry.');
		RETURN;
	END_IF

	iThread := _Plant.iFirstThread;
	iPrevThread := 0;

	WHILE iThread <> 0 DO
		nThreadGuard := nThreadGuard + 1;
		IF nThreadGuard > GUARD THEN
			Plant.Panic(0, 'Thread dispatch failed: thread traversal exceeded GUARD; probable cycle.');
			RETURN;
		END_IF

		IF ValidateInterface(iThread) <> Ok THEN
			Plant.Panic(0, 'Thread dispatch failed: current thread failed ValidateInterface before list access.');
			RETURN;
		END_IF

		iNextThread := iThread.GetNext();

		iCheckThread := iThread.GetPrev();
		IF iCheckThread <> iPrevThread THEN
			Plant.Panic(iThread, 'Thread dispatch failed: current thread _Prev does not match current registry state.');
			RETURN;
		END_IF

		IF iNextThread <> 0 THEN
			IF ValidateInterface(iNextThread) <> Ok THEN
				Plant.Panic(iThread, 'Thread dispatch failed: current thread _Next failed ValidateInterface.');
				RETURN;
			END_IF

			IF iNextThread = iThread THEN
				Plant.Panic(iThread, 'Thread dispatch failed: current thread _Next points to itself.');
				RETURN;
			END_IF

			iCheckThread := iNextThread.GetPrev();
			IF iCheckThread <> iThread THEN
				Plant.Panic(iThread, 'Thread dispatch failed: next thread _Prev does not point back to current thread.');
				RETURN;
			END_IF
		ELSIF _Plant.iLastThread <> iThread THEN
			Plant.Panic(iThread, 'Thread dispatch failed: tail thread does not match _Plant.iLastThread.');
			RETURN;
		END_IF

		iExecute := iThread.GetFirst();
		iLastExecute := iThread.GetLast();
		iPrevExecute := 0;
		nExecuteGuard := 0;

		IF iExecute = 0 THEN
			IF iLastExecute <> 0 THEN
				Plant.Panic(iThread, 'Thread dispatch failed: first execute is 0 but last execute is not 0.');
				RETURN;
			END_IF
		ELSE
			IF ValidateInterface(iLastExecute) <> Ok THEN
				Plant.Panic(iThread, 'Thread dispatch failed: last execute failed ValidateInterface before list access.');
				RETURN;
			END_IF

			iCheckExecute := iExecute.GetPrev();
			IF iCheckExecute <> 0 THEN
				Plant.Panic(iExecute, 'Thread dispatch failed: first execute has a nonzero _Prev link.');
				RETURN;
			END_IF

			iCheckExecute := iLastExecute.GetNext();
			IF iCheckExecute <> 0 THEN
				Plant.Panic(iLastExecute, 'Thread dispatch failed: last execute has a nonzero _Next link.');
				RETURN;
			END_IF
		END_IF

		WHILE iExecute <> 0 DO
			nExecuteGuard := nExecuteGuard + 1;
			IF nExecuteGuard > GUARD THEN
				Plant.Panic(iThread, 'Thread dispatch failed: execute traversal exceeded GUARD; probable cycle.');
				RETURN;
			END_IF

			IF ValidateInterface(iExecute) <> Ok THEN
				Plant.Panic(iThread, 'Thread dispatch failed: current execute failed ValidateInterface before link access.');
				RETURN;
			END_IF

			iNextExecute := iExecute.GetNext();

			iCheckExecute := iExecute.GetPrev();
			IF iCheckExecute <> iPrevExecute THEN
				Plant.Panic(iExecute, 'Thread dispatch failed: current execute _Prev does not match current list state.');
				RETURN;
			END_IF

			IF iNextExecute <> 0 THEN
				IF ValidateInterface(iNextExecute) <> Ok THEN
					Plant.Panic(iExecute, 'Thread dispatch failed: current execute _Next failed ValidateInterface.');
					RETURN;
				END_IF

				IF iNextExecute = iExecute THEN
					Plant.Panic(iExecute, 'Thread dispatch failed: current execute _Next points to itself.');
					RETURN;
				END_IF

				iCheckExecute := iNextExecute.GetPrev();
				IF iCheckExecute <> iExecute THEN
					Plant.Panic(iExecute, 'Thread dispatch failed: next execute _Prev does not point back to current execute.');
					RETURN;
				END_IF
			ELSE
				iCheckExecute := iThread.GetLast();
				IF iCheckExecute <> iExecute THEN
					Plant.Panic(iExecute, 'Thread dispatch failed: tail execute does not match the owning thread last execute.');
					RETURN;
				END_IF
			END_IF

			iExecuteThread := iExecute.GetThread();
			bDefaultedThread := FALSE;
			bMoved := FALSE;

			IF ValidateInterface(iExecuteThread) <> Ok OR NOT Plant._IsThreadRegistered(iExecuteThread) THEN
				iExecuteThread := iMainThread;
				iExecute.SetThread(iMainThread);
				bDefaultedThread := TRUE;

				IF bWarn THEN
					Plant.Warn(iExecute, 'Execute repair: configured _Thread was 0, invalid, or not registered during online-change dispatch; assigned MainThread.');
				END_IF
			END_IF

			IF iExecuteThread <> iThread THEN
				bMoved := TRUE;
				iExecute.SetThread(iThread);
				IF iThread.DetachExecute(iExecute) <> Ok THEN
					Plant.Panic(iExecute, 'Thread dispatch failed: could not detach execute from its current owning thread.');
					RETURN;
				END_IF

				iExecute.SetThread(iExecuteThread);
				IF IsErr(iExecuteThread.AttachExecute(iExecute)) THEN
					Plant.Panic(iExecute, 'Thread dispatch failed: could not attach execute to its configured thread.');
					RETURN;
				END_IF

				IF bWarn AND NOT bDefaultedThread THEN
					Plant.Warn(iExecute, 'Execute dispatch: configured _Thread changed during online change; moved execute to configured thread.');
				END_IF
			END_IF

			IF NOT bMoved THEN
				iPrevExecute := iExecute;
			END_IF
			iExecute := iNextExecute;
		END_WHILE

		iWorker := iThread.GetFirstWorker();
		iLastWorker := iThread.GetLastWorker();
		iPrevWorker := 0;
		nWorkerGuard := 0;

		IF iWorker = 0 THEN
			IF iLastWorker <> 0 THEN
				Plant.Panic(iThread, 'Thread dispatch failed: first worker is 0 but last worker is not 0.');
				RETURN;
			END_IF
		ELSE
			IF ValidateInterface(iLastWorker) <> Ok THEN
				Plant.Panic(iThread, 'Thread dispatch failed: last worker failed ValidateInterface before list access.');
				RETURN;
			END_IF

			iCheckWorker := iWorker.GetPrev();
			IF iCheckWorker <> 0 THEN
				Plant.Panic(iWorker, 'Thread dispatch failed: first worker has a nonzero _Prev link.');
				RETURN;
			END_IF

			iCheckWorker := iLastWorker.GetNext();
			IF iCheckWorker <> 0 THEN
				Plant.Panic(iLastWorker, 'Thread dispatch failed: last worker has a nonzero _Next link.');
				RETURN;
			END_IF
		END_IF

		WHILE iWorker <> 0 DO
			nWorkerGuard := nWorkerGuard + 1;
			IF nWorkerGuard > GUARD THEN
				Plant.Panic(iThread, 'Thread dispatch failed: worker traversal exceeded GUARD; probable cycle.');
				RETURN;
			END_IF

			IF ValidateInterface(iWorker) <> Ok THEN
				Plant.Panic(iThread, 'Thread dispatch failed: current worker failed ValidateInterface before link access.');
				RETURN;
			END_IF

			iNextWorker := iWorker.GetNext();

			iCheckWorker := iWorker.GetPrev();
			IF iCheckWorker <> iPrevWorker THEN
				Plant.Panic(iWorker, 'Thread dispatch failed: current worker _Prev does not match current list state.');
				RETURN;
			END_IF

			IF iNextWorker <> 0 THEN
				IF ValidateInterface(iNextWorker) <> Ok THEN
					Plant.Panic(iWorker, 'Thread dispatch failed: current worker _Next failed ValidateInterface.');
					RETURN;
				END_IF

				IF iNextWorker = iWorker THEN
					Plant.Panic(iWorker, 'Thread dispatch failed: current worker _Next points to itself.');
					RETURN;
				END_IF

				iCheckWorker := iNextWorker.GetPrev();
				IF iCheckWorker <> iWorker THEN
					Plant.Panic(iWorker, 'Thread dispatch failed: next worker _Prev does not point back to current worker.');
					RETURN;
				END_IF
			ELSE
				iCheckWorker := iThread.GetLastWorker();
				IF iCheckWorker <> iWorker THEN
					Plant.Panic(iWorker, 'Thread dispatch failed: tail worker does not match the owning thread last worker.');
					RETURN;
				END_IF
			END_IF

			iWorkerThread := iWorker.GetThread();
			bDefaultedThread := FALSE;
			bMoved := FALSE;

			IF ValidateInterface(iWorkerThread) <> Ok OR NOT Plant._IsThreadRegistered(iWorkerThread) THEN
				iWorkerThread := iMainThread;
				iWorker.SetThread(iMainThread);
				bDefaultedThread := TRUE;

				IF bWarn THEN
					Plant.Warn(iWorker, 'Worker repair: configured Thread was 0, invalid, or not registered during online-change dispatch; assigned MainThread.');
				END_IF
			END_IF

			IF iWorkerThread <> iThread THEN
				bMoved := TRUE;
				iWorker.SetThread(iThread);
				IF iThread.DetachWorker(iWorker) <> Ok THEN
					Plant.Panic(iWorker, 'Thread dispatch failed: could not detach worker from its current owning thread.');
					RETURN;
				END_IF

				iWorker.SetThread(iWorkerThread);
				IF IsErr(iWorkerThread.AttachWorker(iWorker)) THEN
					Plant.Panic(iWorker, 'Thread dispatch failed: could not attach worker to its configured thread.');
					RETURN;
				END_IF

				IF bWarn AND NOT bDefaultedThread THEN
					Plant.Warn(iWorker, 'Worker dispatch: configured Thread changed during online change; moved worker to configured thread.');
				END_IF
			END_IF

			IF NOT bMoved THEN
				iPrevWorker := iWorker;
			END_IF
			iWorker := iNextWorker;
		END_WHILE

		iPrevThread := iThread;
		iThread := iNextThread;
	END_WHILE

	IF _Plant.iFirstWorker = 0 THEN
		IF _Plant.iLastWorker <> 0 THEN
			Plant.Panic(0, 'Thread dispatch failed: first registered worker is 0 but last registered worker is not 0.');
			RETURN;
		END_IF
	ELSE
		IF ValidateInterface(_Plant.iFirstWorker) <> Ok THEN
			Plant.Panic(0, 'Thread dispatch failed: first registered worker failed ValidateInterface before registry access.');
			RETURN;
		END_IF

		IF _Plant.iLastWorker = 0 THEN
			Plant.Panic(0, 'Thread dispatch failed: first registered worker is not 0 but last registered worker is 0.');
			RETURN;
		END_IF

		IF ValidateInterface(_Plant.iLastWorker) <> Ok THEN
			Plant.Panic(0, 'Thread dispatch failed: last registered worker failed ValidateInterface before registry access.');
			RETURN;
		END_IF

		iCheckWorker := _Plant.iFirstWorker.GetPlantPrev();
		IF iCheckWorker <> 0 THEN
			Plant.Panic(_Plant.iFirstWorker, 'Thread dispatch failed: first registered worker has a nonzero _PlantPrev link.');
			RETURN;
		END_IF

		iCheckWorker := _Plant.iLastWorker.GetPlantNext();
		IF iCheckWorker <> 0 THEN
			Plant.Panic(_Plant.iLastWorker, 'Thread dispatch failed: last registered worker has a nonzero _PlantNext link.');
			RETURN;
		END_IF
	END_IF

	iWorker := _Plant.iFirstWorker;
	iPrevWorker := 0;
	nWorkerGuard := 0;

	WHILE iWorker <> 0 DO
		nWorkerGuard := nWorkerGuard + 1;
		IF nWorkerGuard > GUARD THEN
			Plant.Panic(0, 'Thread dispatch failed: registered worker traversal exceeded GUARD; probable cycle.');
			RETURN;
		END_IF

		IF ValidateInterface(iWorker) <> Ok THEN
			Plant.Panic(0, 'Thread dispatch failed: current registered worker failed ValidateInterface before registry access.');
			RETURN;
		END_IF

		iCheckWorker := iWorker.GetPlantPrev();
		IF iCheckWorker <> iPrevWorker THEN
			Plant.Panic(iWorker, 'Thread dispatch failed: current registered worker _PlantPrev does not match current registry state.');
			RETURN;
		END_IF

		iNextWorker := iWorker.GetPlantNext();

		IF iNextWorker <> 0 THEN
			IF ValidateInterface(iNextWorker) <> Ok THEN
				Plant.Panic(iWorker, 'Thread dispatch failed: current registered worker _PlantNext failed ValidateInterface.');
				RETURN;
			END_IF

			IF iNextWorker = iWorker THEN
				Plant.Panic(iWorker, 'Thread dispatch failed: current registered worker _PlantNext points to itself.');
				RETURN;
			END_IF

			iCheckWorker := iNextWorker.GetPlantPrev();
			IF iCheckWorker <> iWorker THEN
				Plant.Panic(iWorker, 'Thread dispatch failed: next registered worker _PlantPrev does not point back to current worker.');
				RETURN;
			END_IF
		ELSIF _Plant.iLastWorker <> iWorker THEN
			Plant.Panic(iWorker, 'Thread dispatch failed: tail registered worker does not match _Plant.iLastWorker.');
			RETURN;
		END_IF

		iWorkerThread := iWorker.GetThread();

		IF ValidateInterface(iWorkerThread) <> Ok OR NOT Plant._IsThreadRegistered(iWorkerThread) THEN
			iWorker.SetThread(iMainThread);

			IF bWarn THEN
				Plant.Warn(iWorker, 'Worker registry repair: configured Thread was 0, invalid, or not registered during online-change dispatch; assigned MainThread.');
			END_IF
		END_IF

		iPrevWorker := iWorker;
		iWorker := iNextWorker;
	END_WHILE

	_ThreadDispatcher := Ok;

__CATCH(_err)
	Plant.Panic(0, 'Thread dispatch failed: exception while repairing or redispatching thread-owned lists.');
	_ThreadDispatcher := Error;
__ENDTRY
END_METHOD

METHOD PRIVATE _ValidatePlant : Result
VAR CONSTANT
	GUARD: UDINT := Param.VALIDATION_GUARD;
END_VAR
VAR
	iEntity: I_Entity;
	iPrevEntity: I_Entity;
	iNextEntity: I_Entity;
	iEntityRaw: I_Generic;
	iMainThread: I_Thread := _Plant.MainThread;
	iThread: I_Thread;
	iPrevThread: I_Thread;
	iNextThread: I_Thread;
	iWorker: I_Worker;
	iPrevWorker: I_Worker;
	iNextWorker: I_Worker;
	iWorkerThread: I_Thread;
	iCheckEntity: I_Entity;
	iCheckThread: I_Thread;
	iCheckWorker: I_Worker;
	bMainThreadFound: BOOL;
	nGuard: UDINT;
	_err: __SYSTEM.ExceptionCode;
END_VAR
_ValidatePlant := Error;

__TRY
	IF ValidateInterface(iMainThread) <> Ok THEN
		Plant.Panic(0, 'Plant validation failed: _Plant.MainThread did not pass ValidateInterface.');
		RETURN;
	END_IF

	IF _Plant.iFirstEntity = 0 THEN
		IF _Plant.iLastEntity <> 0 THEN
			Plant.Panic(0, 'Plant validation failed: first entity is 0 but last entity is not 0.');
			RETURN;
		END_IF
	ELSE
		IF ValidateInterface(_Plant.iFirstEntity) <> Ok THEN
			Plant.Panic(0, 'Plant validation failed: first entity did not pass ValidateInterface.');
			RETURN;
		END_IF

		IF _Plant.iLastEntity = 0 THEN
			Plant.Panic(0, 'Plant validation failed: first entity is not 0 but last entity is 0.');
			RETURN;
		END_IF

		IF ValidateInterface(_Plant.iLastEntity) <> Ok THEN
			Plant.Panic(0, 'Plant validation failed: last entity did not pass ValidateInterface.');
			RETURN;
		END_IF

		iCheckEntity := _Plant.iFirstEntity.GetPrev();
		IF iCheckEntity <> 0 THEN
			Plant.Panic(_Plant.iFirstEntity, 'Plant validation failed: first entity has a nonzero _Prev link.');
			RETURN;
		END_IF

		iCheckEntity := _Plant.iLastEntity.GetNext();
		IF iCheckEntity <> 0 THEN
			Plant.Panic(_Plant.iLastEntity, 'Plant validation failed: last entity has a nonzero _Next link.');
			RETURN;
		END_IF
	END_IF

	iEntity := _Plant.iFirstEntity;
	iPrevEntity := 0;
	nGuard := 0;

	WHILE iEntity <> 0 DO
		nGuard := nGuard + 1;
		IF nGuard > GUARD THEN
			Plant.Panic(0, 'Plant validation failed: entity traversal exceeded GUARD; probable cycle.');
			RETURN;
		END_IF

		IF ValidateInterface(iEntity) <> Ok THEN
			Plant.Panic(0, 'Plant validation failed: current entity did not pass ValidateInterface before link access.');
			RETURN;
		END_IF

		iCheckEntity := iEntity.GetPrev();
		IF iCheckEntity <> iPrevEntity THEN
			Plant.Panic(iEntity, 'Plant validation failed: current entity _Prev does not match previous visited entity.');
			RETURN;
		END_IF

		iEntityRaw := iEntity.GetRaw();
		IF ValidateGeneric(iEntityRaw) <> Ok THEN
			Plant.Panic(iEntity, 'Plant validation failed: current entity _Raw is 0, garbage, or failed generic validation.');
			RETURN;
		END_IF

		iNextEntity := iEntity.GetNext();

		IF iNextEntity <> 0 THEN
			IF ValidateInterface(iNextEntity) <> Ok THEN
				Plant.Panic(iEntity, 'Plant validation failed: current entity _Next did not pass ValidateInterface.');
				RETURN;
			END_IF

			IF iNextEntity = iEntity THEN
				Plant.Panic(iEntity, 'Plant validation failed: current entity _Next points to itself.');
				RETURN;
			END_IF

			iCheckEntity := iNextEntity.GetPrev();
			IF iCheckEntity <> iEntity THEN
				Plant.Panic(iEntity, 'Plant validation failed: next entity _Prev does not point back to current entity.');
				RETURN;
			END_IF
		END_IF

		iPrevEntity := iEntity;
		iEntity := iNextEntity;
	END_WHILE

	IF iPrevEntity <> _Plant.iLastEntity THEN
		Plant.Panic(0, 'Plant validation failed: last visited entity does not match _Plant.iLastEntity.');
		RETURN;
	END_IF

	IF _Plant.iFirstThread = 0 THEN
		IF _Plant.iLastThread <> 0 THEN
			Plant.Panic(0, 'Plant validation failed: first thread is 0 but last thread is not 0.');
			RETURN;
		END_IF
	ELSE
		IF ValidateInterface(_Plant.iFirstThread) <> Ok THEN
			Plant.Panic(0, 'Plant validation failed: first thread did not pass ValidateInterface.');
			RETURN;
		END_IF

		IF _Plant.iLastThread = 0 THEN
			Plant.Panic(0, 'Plant validation failed: first thread is not 0 but last thread is 0.');
			RETURN;
		END_IF

		IF ValidateInterface(_Plant.iLastThread) <> Ok THEN
			Plant.Panic(0, 'Plant validation failed: last thread did not pass ValidateInterface.');
			RETURN;
		END_IF

		iCheckThread := _Plant.iFirstThread.GetPrev();
		IF iCheckThread <> 0 THEN
			Plant.Panic(_Plant.iFirstThread, 'Plant validation failed: first thread has a nonzero _Prev link.');
			RETURN;
		END_IF

		iCheckThread := _Plant.iLastThread.GetNext();
		IF iCheckThread <> 0 THEN
			Plant.Panic(_Plant.iLastThread, 'Plant validation failed: last thread has a nonzero _Next link.');
			RETURN;
		END_IF
	END_IF

	iThread := _Plant.iFirstThread;
	iPrevThread := 0;
	bMainThreadFound := FALSE;
	nGuard := 0;

	WHILE iThread <> 0 DO
		nGuard := nGuard + 1;
		IF nGuard > GUARD THEN
			Plant.Panic(0, 'Plant validation failed: thread traversal exceeded GUARD; probable cycle.');
			RETURN;
		END_IF

		IF ValidateInterface(iThread) <> Ok THEN
			Plant.Panic(0, 'Plant validation failed: current thread did not pass ValidateInterface before link access.');
			RETURN;
		END_IF

		iCheckThread := iThread.GetPrev();
		IF iCheckThread <> iPrevThread THEN
			Plant.Panic(iThread, 'Plant validation failed: current thread _Prev does not match previous visited thread.');
			RETURN;
		END_IF

		IF iThread = iMainThread THEN
			bMainThreadFound := TRUE;
		END_IF

		IF iThread.ValidateThread() <> Ok THEN
			Plant.Panic(iThread, 'Plant validation failed: current thread did not pass ValidateThread.');
			RETURN;
		END_IF

		iNextThread := iThread.GetNext();

		IF iNextThread <> 0 THEN
			IF ValidateInterface(iNextThread) <> Ok THEN
				Plant.Panic(iThread, 'Plant validation failed: current thread _Next did not pass ValidateInterface.');
				RETURN;
			END_IF

			IF iNextThread = iThread THEN
				Plant.Panic(iThread, 'Plant validation failed: current thread _Next points to itself.');
				RETURN;
			END_IF

			iCheckThread := iNextThread.GetPrev();
			IF iCheckThread <> iThread THEN
				Plant.Panic(iThread, 'Plant validation failed: next thread _Prev does not point back to current thread.');
				RETURN;
			END_IF
		END_IF

		iPrevThread := iThread;
		iThread := iNextThread;
	END_WHILE

	IF iPrevThread <> _Plant.iLastThread THEN
		Plant.Panic(0, 'Plant validation failed: last visited thread does not match _Plant.iLastThread.');
		RETURN;
	END_IF

	IF NOT bMainThreadFound THEN
		Plant.Panic(0, 'Plant validation failed: _Plant.MainThread is not linked in the Plant thread registry.');
		RETURN;
	END_IF

	IF _Plant.iFirstWorker = 0 THEN
		IF _Plant.iLastWorker <> 0 THEN
			Plant.Panic(0, 'Plant validation failed: first registered worker is 0 but last registered worker is not 0.');
			RETURN;
		END_IF
	ELSE
		IF ValidateInterface(_Plant.iFirstWorker) <> Ok THEN
			Plant.Panic(0, 'Plant validation failed: first registered worker did not pass ValidateInterface.');
			RETURN;
		END_IF

		IF _Plant.iLastWorker = 0 THEN
			Plant.Panic(0, 'Plant validation failed: first registered worker is not 0 but last registered worker is 0.');
			RETURN;
		END_IF

		IF ValidateInterface(_Plant.iLastWorker) <> Ok THEN
			Plant.Panic(0, 'Plant validation failed: last registered worker did not pass ValidateInterface.');
			RETURN;
		END_IF

		iCheckWorker := _Plant.iFirstWorker.GetPlantPrev();
		IF iCheckWorker <> 0 THEN
			Plant.Panic(_Plant.iFirstWorker, 'Plant validation failed: first registered worker has a nonzero _PlantPrev link.');
			RETURN;
		END_IF

		iCheckWorker := _Plant.iLastWorker.GetPlantNext();
		IF iCheckWorker <> 0 THEN
			Plant.Panic(_Plant.iLastWorker, 'Plant validation failed: last registered worker has a nonzero _PlantNext link.');
			RETURN;
		END_IF
	END_IF

	iWorker := _Plant.iFirstWorker;
	iPrevWorker := 0;
	nGuard := 0;

	WHILE iWorker <> 0 DO
		nGuard := nGuard + 1;
		IF nGuard > GUARD THEN
			Plant.Panic(0, 'Plant validation failed: registered worker traversal exceeded GUARD; probable cycle.');
			RETURN;
		END_IF

		IF ValidateInterface(iWorker) <> Ok THEN
			Plant.Panic(0, 'Plant validation failed: current registered worker did not pass ValidateInterface before registry access.');
			RETURN;
		END_IF

		iCheckWorker := iWorker.GetPlantPrev();
		IF iCheckWorker <> iPrevWorker THEN
			Plant.Panic(iWorker, 'Plant validation failed: current registered worker _PlantPrev does not match previous visited worker.');
			RETURN;
		END_IF

		iWorkerThread := iWorker.GetThread();
		IF ValidateInterface(iWorkerThread) <> Ok THEN
			Plant.Panic(iWorker, 'Plant validation failed: current registered worker Thread is 0 or failed ValidateInterface.');
			RETURN;
		END_IF

		IF NOT Plant._IsThreadRegistered(iWorkerThread) THEN
			Plant.Panic(iWorker, 'Plant validation failed: current registered worker Thread is not linked in the Plant thread registry.');
			RETURN;
		END_IF

		iNextWorker := iWorker.GetPlantNext();

		IF iNextWorker <> 0 THEN
			IF ValidateInterface(iNextWorker) <> Ok THEN
				Plant.Panic(iWorker, 'Plant validation failed: current registered worker _PlantNext did not pass ValidateInterface.');
				RETURN;
			END_IF

			IF iNextWorker = iWorker THEN
				Plant.Panic(iWorker, 'Plant validation failed: current registered worker _PlantNext points to itself.');
				RETURN;
			END_IF

			iCheckWorker := iNextWorker.GetPlantPrev();
			IF iCheckWorker <> iWorker THEN
				Plant.Panic(iWorker, 'Plant validation failed: next registered worker _PlantPrev does not point back to current worker.');
				RETURN;
			END_IF
		END_IF

		iPrevWorker := iWorker;
		iWorker := iNextWorker;
	END_WHILE

	IF iPrevWorker <> _Plant.iLastWorker THEN
		Plant.Panic(0, 'Plant validation failed: last visited registered worker does not match _Plant.iLastWorker.');
		RETURN;
	END_IF

	_ValidatePlant := Ok;

__CATCH(_err)
	Plant.Panic(0, 'Plant validation failed: exception while reading validation interfaces or links.');
	_ValidatePlant := Error;
__ENDTRY
END_METHOD

// TRUE while Plant is running startup initialization.
PROPERTY IsInit : BOOL
GET
IsInit := _Plant.bInit;
END_GET
END_PROPERTY

// Advances iEntity to next registered entity; returns Ok found, None end, Error invalid ref.
METHOD NextEtt : Result
VAR_INPUT
	iEntity: REFERENCE TO I_Entity; // Iterator variable; set to 0 before first call.
END_VAR
IF NOT __ISVALIDREF(iEntity) THEN
	NextEtt := Error;
	RETURN;
END_IF

IF iEntity = 0 THEN
	iEntity := _Plant.iFirstEntity;
ELSE
	iEntity := iEntity.GetNext();
END_IF

IF iEntity <> 0 THEN
	NextEtt := Ok;
ELSE
	NextEtt := None;
END_IF
END_METHOD

// Records a panic; startup panics stop cyclic execution after init.
METHOD Panic
VAR_INPUT
	iSource: I_Debug; // Source object for diagnostics; may be 0.
	sComment: Str; // Short diagnostic message.
END_VAR
IF _Plant.nLastPanic > Param.MAX_PANIC_MSG THEN
	_Plant.nTotalPanic := _Plant.nTotalPanic + 1;
	RETURN;


ELSIF _Plant.nLastPanic = Param.MAX_PANIC_MSG THEN
	_Plant.panic[_Plant.nLastPanic].iSource := 0;
	_Plant.panic[_Plant.nLastPanic].sComment := 'Panics buffer overflow!';

	_Plant.nLastPanic := _Plant.nLastPanic + 1;
	_Plant.nTotalPanic := _Plant.nTotalPanic + 1;
	RETURN;

END_IF

_Plant.panic[_Plant.nLastPanic].iSource := iSource;
_Plant.panic[_Plant.nLastPanic].sComment := sComment;
_Plant.nLastPanic := _Plant.nLastPanic + 1;
_Plant.nTotalPanic := _Plant.nTotalPanic + 1;
END_METHOD

// Fixed-size panic message buffer.
PROPERTY PanicArr : ARRAY[1..PARAM.MAX_PANIC_MSG] OF DebugStruct;
GET
PanicArr := _Plant.panic;
END_GET
END_PROPERTY

// TRUE after at least one panic has been recorded.
PROPERTY Panicked : BOOL
GET
Panicked := _Plant.nTotalPanic <> 0;
END_GET
END_PROPERTY

// Moves iEntity to previous registered entity; returns Ok found, None end, Error invalid ref.
METHOD PrevEtt : Result
VAR_INPUT
	iEntity: REFERENCE TO I_Entity; // Iterator variable; set to 0 before first call.
END_VAR
IF NOT __ISVALIDREF(iEntity) THEN
	PrevEtt := Error;
	RETURN;
END_IF

IF iEntity = 0 THEN
	iEntity := _Plant.iLastEntity;
ELSE
	iEntity := iEntity.GetPrev();
END_IF

IF iEntity <> 0 THEN
	PrevEtt := Ok;
ELSE
	PrevEtt := None;
END_IF
END_METHOD

// Runs startup once, then main thread each cycle; cyclic work stops after startup panic.
METHOD Run
IF _Plant.bInit THEN
	IF _Plant.bPanic THEN
		RETURN;
	END_IF

	IF _ThreadDispatcher(bWarn := FALSE) <> Ok THEN
		_Plant.bPanic := TRUE;
		RETURN;
	END_IF
	
	_CallPreInits();
	_CallInits();
	_CallPostInits();
	_ClearNewInstanceFlags();


	IF Panicked THEN
		Tc2_System.ADSLOGSTR(Tc2_System.ADSLOG_MSGTYPE_ERROR, Tc2_Standard.CONCAT('Runtime disabled! Total Panic: ', UDINT_TO_STRING(_Plant.nTotalPanic)), '');
		_Plant.bPanic := TRUE;
	END_IF

	IF _Plant.nTotalWarn > 0 THEN
		Tc2_System.ADSLOGSTR(Tc2_System.ADSLOG_MSGTYPE_WARN, Tc2_Standard.CONCAT('Total warnings: ', UDINT_TO_STRING(_Plant.nTotalWarn)), '');
	END_IF

	_Plant.bOnlineChangeEntityCreated := FALSE;
	_Plant.bOnlineChangeEntityDeleted := FALSE;
	_Plant.bOnlineChange := FALSE;

	_Plant.bInit := FALSE;
	RETURN;
END_IF

IF _Plant.bOnlineChange THEN
	IF _ThreadDispatcher(bWarn := TRUE) <> Ok THEN
		_Plant.bPanic := TRUE;
		RETURN;
	END_IF

	IF _ValidatePlant() <> Ok THEN
		_Plant.bPanic := TRUE;
		RETURN;
	END_IF

	IF _Plant.bOnlineChangeEntityCreated THEN
		_CallPreInits();
		_CallInits();
		_CallPostInits();

		IF Panicked THEN
			_Plant.bPanic := TRUE;
			_Plant.bOnlineChangeEntityCreated := FALSE;
			_Plant.bOnlineChangeEntityDeleted := FALSE;
			_Plant.bOnlineChange := FALSE;
			RETURN;
		END_IF
	END_IF

	_CallOnlineChange();
	_ClearNewInstanceFlags();

	_Plant.bOnlineChangeEntityCreated := FALSE;
	_Plant.bOnlineChangeEntityDeleted := FALSE;
	_Plant.bOnlineChange := FALSE;
END_IF

_Plant.MainThread.Run();
END_METHOD

// Total number of recorded panic attempts.
PROPERTY TotalPanic : UDINT
GET
TotalPanic := _Plant.nTotalPanic;
END_GET
END_PROPERTY

// Total number of recorded warning attempts.
PROPERTY TotalWarn : UDINT
GET
TotalWarn := _Plant.nTotalWarn;
END_GET
END_PROPERTY

METHOD ValidateGeneric : Result
VAR_INPUT
	iToValidate: I_Generic;
END_VAR
VAR
	_err: __SYSTEM.ExceptionCode;
	_iValidate: _I_ValidateGeneric;
END_VAR
IF iToValidate = 0 THEN
	ValidateGeneric := Error;
	RETURN;
END_IF

__TRY
	__QUERYINTERFACE(iToValidate, _iValidate);
	ValidateGeneric := Ok;
__CATCH(_err)
	ValidateGeneric := Error;
__ENDTRY
END_METHOD

METHOD ValidateInterface : Result
VAR_INPUT
	iToValidate: I_ValidateInterface;
END_VAR
VAR
	_err: __SYSTEM.ExceptionCode;
END_VAR
IF iToValidate = 0 THEN
	ValidateInterface := Error;
	RETURN;
END_IF

__TRY
	iToValidate.ValidateInterface();
	ValidateInterface := Ok;
__CATCH(_err)
	ValidateInterface := Error;
__ENDTRY
END_METHOD

// Records a warning without stopping cyclic execution.
METHOD Warn
VAR_INPUT
	iSource: I_Debug; // Source object for diagnostics; may be 0.
	sComment: Str; // Short diagnostic message.
END_VAR
IF _Plant.nLastWarn > Param.MAX_WARN_MSG THEN
	_Plant.nTotalWarn := _Plant.nTotalWarn + 1;
	RETURN;


ELSIF _Plant.nLastWarn = Param.MAX_WARN_MSG THEN
	_Plant.warn[_Plant.nLastWarn].iSource := 0;
	_Plant.warn[_Plant.nLastWarn].sComment := 'Warnings buffer overflow!';

	_Plant.nLastWarn := _Plant.nLastWarn + 1;
	_Plant.nTotalWarn := _Plant.nTotalWarn + 1;
	RETURN;

END_IF

_Plant.warn[_Plant.nLastWarn].iSource := iSource;
_Plant.warn[_Plant.nLastWarn].sComment := sComment;
_Plant.nLastWarn := _Plant.nLastWarn + 1;
_Plant.nTotalWarn := _Plant.nTotalWarn + 1;
END_METHOD

// Fixed-size warning message buffer.
PROPERTY WarnArr : ARRAY[1..PARAM.MAX_WARN_MSG] OF DebugStruct;
GET
WarnArr := _Plant.warn;
END_GET
END_PROPERTY

END_PROGRAM

// ---- Plant/Entity/Entity.TcPOU
// Registers an I_Generic owner in the global entity list.
FUNCTION_BLOCK FINAL Entity IMPLEMENTS I_Entity
VAR
	{attribute 'no_copy'}
	{attribute 'no_init'}
	_iGeneric: I_Generic;	
	_iNext: I_Entity;
	_iPrev: I_Entity;
	_eResult: Result;
	_bNewInstance: BOOL;
END_VAR

METHOD INTERNAL GetNext : I_Entity
GetNext := _iNext;
END_METHOD

METHOD INTERNAL SetNext
VAR_INPUT
	iNext: I_Entity;
END_VAR
_iNext := iNext;
END_METHOD

METHOD INTERNAL GetPrev : I_Entity
GetPrev := _iPrev;
END_METHOD

METHOD INTERNAL SetPrev
VAR_INPUT
	iPrev: I_Entity;
END_VAR
_iPrev := iPrev;
END_METHOD

METHOD INTERNAL GetRaw : I_Generic
GetRaw := _iGeneric;
END_METHOD

METHOD INTERNAL SetRaw
VAR_INPUT
	iRaw: I_Generic;
END_VAR
_iGeneric := iRaw;
END_METHOD

PROPERTY INTERNAL _Result : Result
GET
_Result := _eResult;
END_GET
END_PROPERTY

PROPERTY INTERNAL _NewInstance : BOOL
GET
_NewInstance := _bNewInstance;
END_GET
SET
_bNewInstance := _NewInstance;
END_SET
END_PROPERTY

//FB_Exit must be implemented explicitly. If there is an implementation, then the
//method is called before the controller removes the code of the function block instance
//(implicit call). The return value is not evaluated.
{attribute 'hide'}
METHOD FB_Exit: BOOL
VAR_INPUT
    bInCopyCode: BOOL;  // TRUE: the exit method is called in order to leave the instance which will be copied afterwards (online change).  
END_VAR
IF NOT bInCopyCode THEN
	IF Plant._DetachEntity(THIS^) = Ok THEN
		_Plant.bOnlineChangeEntityDeleted := TRUE;
	END_IF
END_IF
END_METHOD

// Registers iGeneric during initialization; panics if iGeneric is 0.
{attribute 'hide'}
METHOD FB_Init: BOOL
VAR_INPUT
    bInitRetains: BOOL; // TRUE on retain initialization.
    bInCopyCode: BOOL;  // TRUE before online-change copy.
	iGeneric: I_Generic; // Owner to register; must not be 0.
END_VAR
IF iGeneric = 0 THEN
	_eResult := Error;
	Plant.Panic(THIS^, 'Entity cannot be initialized with 0');
	RETURN;

END_IF

_iGeneric := iGeneric;

IF _eResult <> None THEN
	RETURN;
END_IF

IF (_eResult := Plant._AttachEntity(THIS^)) = Ok THEN
	_bNewInstance := TRUE;
	_Plant.bOnlineChangeEntityCreated := TRUE;
ELSE
	Plant.Panic(THIS^, __POUNAME());
END_IF
END_METHOD

// Raw discoverable interface for __QUERYINTERFACE.
PROPERTY Raw : I_Generic
GET
Raw := _iGeneric;
END_GET
END_PROPERTY

{attribute 'hide'}
METHOD ValidateInterface
END_METHOD

END_FUNCTION_BLOCK

// ---- Utils/Result/IsSome.TcPOU
// TRUE when nIn <> 0; copies nIn to nOut.
FUNCTION IsSome : BOOL
VAR_INPUT
    nIn : Result; // Result to test.
END_VAR
VAR_OUTPUT
    nOut : Result; // Copy of nIn.
END_VAR

IsSome := nIn <> 0;
nOut := nIn;

END_FUNCTION

// ---- Plant/Job/Worker.TcPOU
// Registers an I_Job owner as a startable worker.
FUNCTION_BLOCK FINAL Worker IMPLEMENTS I_Worker, I_ValidateInterface
VAR
	_iThread: I_Thread := _Plant.MainThread;
	{attribute 'no_copy'}
	{attribute 'no_init'}
	_iJob: I_Job;
	_iNext: I_Worker;
	_iPrev: I_Worker;
	_iPlantNext: I_Worker;
	_iPlantPrev: I_Worker;
	_eState: JobState;
END_VAR

METHOD INTERNAL GetNext : I_Worker
GetNext := _iNext;
END_METHOD

METHOD INTERNAL SetNext
VAR_INPUT
	iNext: I_Worker;
END_VAR
_iNext := iNext;
END_METHOD

METHOD INTERNAL GetPlantNext : I_Worker
GetPlantNext := _iPlantNext;
END_METHOD

METHOD INTERNAL SetPlantNext
VAR_INPUT
	iNext: I_Worker;
END_VAR
_iPlantNext := iNext;
END_METHOD

METHOD INTERNAL GetPlantPrev : I_Worker
GetPlantPrev := _iPlantPrev;
END_METHOD

METHOD INTERNAL SetPlantPrev
VAR_INPUT
	iPrev: I_Worker;
END_VAR
_iPlantPrev := iPrev;
END_METHOD

METHOD INTERNAL GetPrev : I_Worker
GetPrev := _iPrev;
END_METHOD

METHOD INTERNAL SetPrev
VAR_INPUT
	iPrev: I_Worker;
END_VAR
_iPrev := iPrev;
END_METHOD

METHOD INTERNAL GetThread : I_Thread
GetThread := _iThread;
END_METHOD

METHOD INTERNAL SetThread
VAR_INPUT
	iThread: I_Thread;
END_VAR
_iThread := iThread;
END_METHOD

//FB_Exit must be implemented explicitly. If there is an implementation, then the
//method is called before the controller removes the code of the function block instance
//(implicit call). The return value is not evaluated.
{attribute 'hide'}
METHOD FB_Exit: BOOL
VAR_INPUT
    bInCopyCode: BOOL;  // TRUE: the exit method is called in order to leave the instance which will be copied afterwards (online change).
END_VAR
IF NOT bInCopyCode THEN
	IF Plant.ValidateInterface(_iThread) = Ok THEN
		_iThread.DetachWorker(THIS^);
	END_IF

	Plant._DetachWorker(THIS^);
END_IF
END_METHOD

// Registers iJob; panics if iJob is 0.
{attribute 'hide'}
METHOD FB_Init: BOOL
VAR_INPUT
    bInitRetains: BOOL; // TRUE on retain initialization.
    bInCopyCode: BOOL;  // TRUE before online-change copy.

	iJob			: I_Job; // Job owner; must not be 0.
END_VAR
IF _iJob = 0 THEN
	IF iJob = 0 THEN
		Plant.Panic(THIS^, Tc2_Standard.CONCAT(__POUNAME(), ': Itf = 0!'));
		RETURN;
	END_IF

	_iJob := iJob;
END_IF

IF bInCopyCode THEN
	RETURN;
END_IF

IF IsErr(Plant._AttachWorker(THIS^)) THEN
	Plant.Panic(THIS^, 'Worker initialization failed: could not attach worker to Plant registry.');
END_IF
END_METHOD

METHOD INTERNAL Process
VAR_OUTPUT
	iNext: I_Worker;
END_VAR
CASE _eState OF
	JobState.Init:
		_iJob.JobInit();
		_eState := JobState.Busy;
		iNext := _iNext;

	JobState.Busy:
		_iJob.JobExecute();
		iNext := _iNext;

	JobState.Done:
		iNext := _iNext;
		IF IsOk(_iThread.DetachWorker(THIS^)) THEN
			_iJob.JobExit();
			_eState := JobState.Idle;
		END_IF

END_CASE
END_METHOD

// Starts idle job; returns Ok attached, None command busy, Error invalid state or job.
METHOD Start : Result
VAR_INPUT
END_VAR
IF _iJob = 0 THEN
	Start := Error;
	RETURN;
END_IF

CASE _eState OF
	JobState.Init:
		Start := Error;

	JobState.Idle:
		_eState := JobState.Init;
		Start := _iThread.AttachWorker(THIS^);

	JobState.Busy:
		Start := Error;

	JobState.Done:
		Start := Error;

END_CASE
END_METHOD

// Current worker state.
PROPERTY State : JobState
GET
State := _eState;
END_GET
END_PROPERTY

// Requests stop; Busy moves to Done and calls JobExit before returning Idle.
METHOD Stop
VAR_INPUT
END_VAR
_eState := JobState.Done;
END_METHOD

// Thread that processes this worker; can change while Idle.
PROPERTY Thread : I_Thread
GET
Thread := _iThread;
END_GET
SET
IF _eState = JobState.Idle THEN
	IF Plant.IsInit THEN
		_iThread := Thread;
		RETURN;
	END_IF

	IF Plant.ValidateInterface(Thread) <> Ok OR NOT Plant._IsThreadRegistered(Thread) THEN
		Plant.Warn(THIS^, 'Worker thread assignment repair: configured Thread was 0, invalid, or not registered; assigned MainThread.');
		_iThread := _Plant.MainThread;
		RETURN;
	END_IF

	_iThread := Thread;
END_IF
END_SET
END_PROPERTY

METHOD ValidateInterface
VAR_INPUT
END_VAR
END_METHOD

END_FUNCTION_BLOCK

// ---- Utils/Result/IsErr.TcPOU
// TRUE when nIn < 0; copies nIn to nOut.
FUNCTION IsErr : BOOL
VAR_INPUT
    nIn : Result; // Result to test.
END_VAR
VAR_OUTPUT
    nOut : Result; // Copy of nIn.
END_VAR

IsErr := nIn < 0;
nOut := nIn;

END_FUNCTION

// ---- Utils/Result/IsOk.TcPOU
// TRUE when nIn > 0; copies nIn to nOut.
FUNCTION IsOk : BOOL
VAR_INPUT
    nIn : Result; // Result to test.
END_VAR
VAR_OUTPUT
    nOut : Result; // Copy of nIn.
END_VAR

IsOk := nIn > 0;
nOut := nIn;

END_FUNCTION

// ---- Plant/Execute/Execute.TcPOU
// Registers an I_Execute owner for cyclic execution.
FUNCTION_BLOCK FINAL Execute IMPLEMENTS _I_Execute, I_Debug, I_ValidateInterface
VAR
	_iThread: I_Thread := _Plant.MainThread;
	{attribute 'no_copy'}
	{attribute 'no_init'}
	_iExecute: I_Execute;
	_iPrev: _I_Execute;
	_iNext: _I_Execute;
END_VAR

METHOD INTERNAL _Exe
VAR_OUTPUT
	iNext: _I_Execute;
END_VAR
_iExecute.Execute();
iNext := _iNext;
END_METHOD

METHOD INTERNAL GetNext : _I_Execute
GetNext := _iNext;
END_METHOD

METHOD INTERNAL SetNext
VAR_INPUT
	iNext: _I_Execute;
END_VAR
_iNext := iNext;
END_METHOD

METHOD INTERNAL GetPrev : _I_Execute
GetPrev := _iPrev;
END_METHOD

METHOD INTERNAL SetPrev
VAR_INPUT
	iPrev: _I_Execute;
END_VAR
_iPrev := iPrev;
END_METHOD

METHOD INTERNAL GetThread : I_Thread
GetThread := _iThread;
END_METHOD

METHOD INTERNAL SetThread
VAR_INPUT
	iThread: I_Thread;
END_VAR
_iThread := iThread;
END_METHOD

//FB_Exit must be implemented explicitly. If there is an implementation, then the
//method is called before the controller removes the code of the function block instance
//(implicit call). The return value is not evaluated.
{attribute 'hide'}
METHOD FB_Exit: BOOL
VAR_INPUT
    bInCopyCode: BOOL;  // TRUE: the exit method is called in order to leave the instance which will be copied afterwards (online change).  
END_VAR
IF NOT bInCopyCode THEN
	_iThread.DetachExecute(THIS^);
END_IF
END_METHOD

// Registers iExecute during initialization; panics if iExecute is 0.
{attribute 'hide'}
METHOD FB_Init: BOOL
VAR_INPUT
    bInitRetains: BOOL; // TRUE on retain initialization.
    bInCopyCode: BOOL;  // TRUE before online-change copy.
	
	iExecute			: I_Execute; // Owner to execute cyclically; must not be 0.
END_VAR
IF (_iExecute := iExecute) = 0 THEN
	Plant.Panic(THIS^, Tc2_Standard.CONCAT(__POUNAME(), ': Itf = 0!'));
	RETURN;
END_IF

IF bInCopyCode THEN
	RETURN;
END_IF

_iThread := _Plant.MainThread;
_Plant.MainThread.AttachExecute(THIS^);
END_METHOD

// Thread that runs this executor; set during initialization.
PROPERTY Thread : I_Thread
GET
Thread := _iThread;
END_GET
SET
IF NOT Plant.IsInit THEN
	RETURN;
END_IF

_iThread := Thread;
END_SET
END_PROPERTY

{attribute 'hide'}
METHOD ValidateInterface
END_METHOD

END_FUNCTION_BLOCK

// ---- Utils/Color/Argbb.TcPOU
// ARGB component builder.
FUNCTION_BLOCK Argbb
VAR
	_r: BYTE;
	_g: BYTE;
	_b: BYTE;
	_a: BYTE;
END_VAR

// Alpha channel.
PROPERTY Alpha : BYTE
GET
Alpha := _a;
END_GET
SET
_a := Alpha;
END_SET
END_PROPERTY

// Blue channel.
PROPERTY Blue : BYTE
GET
Blue := _b;
END_GET
SET
_b := Blue;
END_SET
END_PROPERTY

// Green channel.
PROPERTY Green : BYTE
GET
Green := _g;
END_GET
SET
_g := Green;
END_SET
END_PROPERTY

// Packed ARGB value.
PROPERTY Raw : Argb
GET
Raw := 	USINT_TO_UDINT(_b) OR
			SHL(USINT_TO_UDINT(_g), 8) OR
			SHL(USINT_TO_UDINT(_r), 16) OR
			SHL(USINT_TO_UDINT(_a), 24);
END_GET
SET
_b := UDINT_TO_USINT(Raw AND 16#FF);
_g := UDINT_TO_USINT(SHR(Raw, 8) AND 16#FF);
_r := UDINT_TO_USINT(SHR(Raw, 16) AND 16#FF);
_a := UDINT_TO_USINT(SHR(Raw, 24) AND 16#FF);
END_SET
END_PROPERTY

// Red channel.
PROPERTY Red : BYTE
GET
Red := _r;
END_GET
SET
_r := Red;
END_SET
END_PROPERTY

// Sets all color channels.
METHOD Set
VAR_INPUT
	nRed: USINT; // Red channel.
	nGreen: USINT; // Green channel.
	nBlue: USINT; // Blue channel.
	nAlpha: USINT; // Alpha channel.
END_VAR
_r := nRed;
_g := nGreen;
_b := nBlue;
_a := nAlpha;
END_METHOD

END_FUNCTION_BLOCK

// ---- Utils/Color/GenArgb.TcPOU
// Packs color components into ARGB.
FUNCTION GenArgb : Argb
VAR_INPUT
	nRed: USINT; // Red channel.
	nGreen: USINT; // Green channel.
	nBlue: USINT; // Blue channel.
	nAlpha: USINT; // Alpha channel.
END_VAR

GenArgb := USINT_TO_UDINT(nBlue) OR
			SHL(USINT_TO_UDINT(nGreen), 8) OR
			SHL(USINT_TO_UDINT(nRed), 16) OR
			SHL(USINT_TO_UDINT(nAlpha), 24);

END_FUNCTION

// ---- Utils/Math/Math.TcPOU
// Numeric helper namespace.
PROGRAM Math
VAR
END_VAR

// Time-compensated smoothing coefficient clamped to 0..1.
METHOD ExptDecay : LREAL
VAR_INPUT
    rBlendFactor : LREAL;   // Base blend factor, clamped 0..1.
    rDeltaTime   : LREAL := 0.01;   // Sample time in seconds.
END_VAR
rBlendFactor := LIMIT(0.0, rBlendFactor, 1.0);
rDeltaTime   := MAX(rDeltaTime, 0.0);
ExptDecay := LIMIT(0.0, 1.0 - EXPT(1.0 - rBlendFactor, rDeltaTime), 1.0);
END_METHOD

// Low-pass coefficient from cutoff frequency; clamped to 0..1.
METHOD FreqCutoffCoef : LREAL
VAR_STAT CONSTANT
	rA: LREAL := 2.0 * 3.141592653589793;
END_VAR
VAR_INPUT
    rCutoffHz  : LREAL;   // Cutoff frequency in Hz.
    rDeltaTime : LREAL;   // Sample time in seconds.
END_VAR
VAR
	rOmega : LREAL;
END_VAR
rCutoffHz  := MAX(rCutoffHz, 0.0);
rDeltaTime := MAX(rDeltaTime, 0.0);
rOmega := rA * rCutoffHz;
FreqCutoffCoef := 1.0 - EXP(-rOmega * rDeltaTime);
FreqCutoffCoef := LIMIT(0.0, FreqCutoffCoef, 1.0);
END_METHOD

// Scales rX from input range to output range; returns 0 when input span is 0.
METHOD LinearScale : LREAL
VAR_INPUT
	rX				: LREAL; // Input value.
	rMinX			: LREAL; // Input range minimum.
	rMaxX			: LREAL; // Input range maximum.
	rMinY			: LREAL := 0; // Output range minimum.
	rMaxY			: LREAL := 1; // Output range maximum.
END_VAR
VAR
	_rDnmtr			: LREAL := rMaxX - rMinX;
END_VAR
IF _rDnmtr <> 0 THEN
	LinearScale := rMinY + ((rX - rMinX)/_rDnmtr) * (rMaxY - rMinY);
END_IF
END_METHOD

// First-order filter output.
METHOD LowPassFilter : LREAL
VAR_INPUT
	rX				: LREAL; // New input.
	rPrvY			: LREAL; // Previous output.
	
	rCoefficient	: LREAL; // Blend coefficient, normally 0..1.
END_VAR
LowPassFilter := rX * rCoefficient + rPrvY * (1 - rCoefficient);
END_METHOD

// Returns pseudo-random LREAL.
METHOD Random : LREAL
VAR_STAT
	_nSeed		: INT;
END_VAR
VAR
	_drand		: Tc2_System.DRAND;
END_VAR
_drand(Seed := _nSeed, Num => Random);
_nSeed := _nSeed + 1;
END_METHOD

// Rounds rValue at decimal position nPosition.
METHOD Round : LREAL
VAR_INPUT
	rValue: LREAL; // Value to round.
	nPosition: SINT; // Decimal position.
END_VAR
VAR
	rFactor: LREAL := 0;
	rTemp: LINT := 0;
END_VAR
rFactor := EXPT(10, -nPosition);
rTemp := LREAL_TO_LINT(rValue * rFactor);
Round := LINT_TO_LREAL(rTemp) / rFactor;
END_METHOD

END_PROGRAM

// ---- Utils/Path/Path.TcPOU
// Builds a slash-delimited path from the TwinCAT instance path.
{attribute 'reflection'}
FUNCTION_BLOCK Path IMPLEMENTS I_Path
VAR
	{attribute 'instance-path'} 
    {attribute 'noinit'}
	_sPath			: Str;
	
	_nLength		: USINT;
	_nOptionPos		: USINT;
	_nOptionLen		: USINT;
END_VAR

{attribute 'hide'}
METHOD FB_init : BOOL
VAR_INPUT
	bInitRetains : BOOL; // if TRUE, the retain variables are initialized (warm start / cold start)
	bInCopyCode : BOOL;  // if TRUE, the instance afterwards gets moved into the copy code (online change)
END_VAR
VAR
	i				: INT;
	_sChar			: Ch;
END_VAR
// Delete this name segment
FOR i := Tc2_Standard.LEN(_sPath) TO 1 BY -1 DO
	IF Tc2_Standard.MID(_sPath, 1, i) = '.' THEN
		_sPath := Tc2_Standard.LEFT(_sPath, i - 1);
		EXIT;
	END_IF
END_FOR

// Delete solution segment
_sPath := Tc2_Standard.RIGHT(_sPath, Tc2_Standard.LEN(_sPath) - Tc2_Standard.FIND(_sPath, '.'));
// Delete project segment
_sPath := Tc2_Standard.RIGHT(_sPath, Tc2_Standard.LEN(_sPath) - Tc2_Standard.FIND(_sPath, '.'));

// Replace '[' with '.' and remove ']' 
FOR i := 1 TO Tc2_Standard.LEN(_sPath) DO
	_sChar := Tc2_Standard.MID(_sPath, 1, i);
	IF _sChar = '[' THEN
		_sPath := Tc2_Standard.REPLACE(_sPath, '.', 1, i);
	ELSIF _sChar = ']' THEN
		_sPath := Tc2_Standard.DELETE(_sPath, 1, i);
	END_IF
END_FOR

// Replace dots
FOR i := 1 TO Tc2_Standard.LEN(_sPath) DO
	_sChar := Tc2_Standard.MID(_sPath, 1, i);
	IF _sChar = '.' THEN
		_sPath := Tc2_Standard.REPLACE(_sPath, '/', 1, i);
	END_IF
END_FOR
_sPath := Tc2_Standard.CONCAT('/', _sPath);
_nLength := INT_TO_USINT(Tc2_Standard.LEN(_sPath));
END_METHOD

// Full generated path including options.
PROPERTY Get : Str
GET
Get := _sPath;
END_GET
END_PROPERTY

// TRUE when the path contains sSegment.
METHOD Has : BOOL
VAR_INPUT
	sSegment: Str; // Segment to find.
END_VAR
VAR
	i: USINT;
	c: Ch;
	nSegLen: USINT := 0;
	nSegPos: USINT := 1;
END_VAR
FOR i := 1 TO _nLength DO
	c := Tc2_Standard.MID(_sPath, 1, i);
	IF (c = '/') OR (c = '=') OR (c = '?') OR (c = '&') THEN
		IF Tc2_Standard.MID(_sPath, nSegLen, nSegPos) = sSegment THEN
			Has := TRUE;
			RETURN;
		END_IF
		
		nSegPos := i + 1;
		nSegLen := 0;
	ELSE
		nSegLen := nSegLen + 1;
	END_IF
END_FOR

IF Tc2_Standard.MID(_sPath, nSegLen, nSegPos) = sSegment THEN
	Has := TRUE;
	RETURN;
END_IF
END_METHOD

// Full path length including options.
PROPERTY Length : USINT
GET
Length := _nLength + _nOptionLen;
END_GET
END_PROPERTY

// Generated path without options.
PROPERTY Name : Str
GET
IF _nOptionPos <> 0 THEN
	Name := Tc2_Standard.LEFT(_sPath, _nOptionPos);
ELSE
	Name := Tc2_Standard.LEFT(_sPath, _nLength);
END_IF
END_GET
END_PROPERTY

// Optional query-style path segment.
PROPERTY Option : Str
GET
VAR
	i				: INT;
END_VAR
IF _nOptionPos <> 0 THEN
	Option := Tc2_Standard.DELETE(_sPath, _nOptionPos, 1);
ELSE
	Option := '';
END_IF
END_GET
SET
IF Option <> '' THEN
    _nOptionLen := INT_TO_USINT(Tc2_Standard.LEN(Option));    
    IF _nOptionPos <> 0 THEN
        _sPath := Tc2_Standard.LEFT(_sPath, _nOptionPos);
        _sPath := Tc2_Standard.CONCAT(_sPath, Option);
		
    ELSE
        // The option does not exist, so we append it
		_nLength := _nLength + _nOptionLen;
        _nOptionPos := INT_TO_USINT(Tc2_Standard.LEN(_sPath) + 1);
        _sPath := Tc2_Standard.CONCAT(_sPath, '?');
        _sPath := Tc2_Standard.CONCAT(_sPath, Option);
		
    END_IF
	
ELSIF _nOptionPos <> 0 THEN
    _sPath := Tc2_Standard.LEFT(_sPath, _nOptionPos - 1);
	_nLength := _nLength - _nOptionLen;
	_nOptionLen := 0;
    _nOptionPos := 0;
	
END_IF
END_SET
END_PROPERTY

END_FUNCTION_BLOCK

// ---- Utils/Result/IsFail.TcPOU
// TRUE when nIn <= 0; copies nIn to nOut.
FUNCTION IsFail : BOOL
VAR_INPUT
    nIn : Result; // Result to test.
END_VAR
VAR_OUTPUT
    nOut : Result; // Copy of nIn.
END_VAR

IsFail := nIn <= 0;
nOut := nIn;

END_FUNCTION

// ---- Utils/Result/IsNone.TcPOU
// TRUE when nIn = 0; copies nIn to nOut.
FUNCTION IsNone : BOOL
VAR_INPUT
    nIn : Result; // Result to test.
END_VAR
VAR_OUTPUT
    nOut : Result; // Copy of nIn.
END_VAR

IsNone := nIn = 0;
nOut := nIn;

END_FUNCTION

// ---- Utils/Strings/Strb/Strb.TcPOU
// Chainable 255-character string builder.
FUNCTION_BLOCK FINAL Strb IMPLEMENTS I_Strb
VAR
	_sString	: Str;
	_nLength	: INT;
END_VAR

PROPERTY PRIVATE _this : I_Strb
GET
VAR
	_iThis : I_Strb := THIS^;
END_VAR
_this := _iThis;
END_GET
END_PROPERTY

// Appends text; truncates at 255 chars.
METHOD Append : I_Strb
VAR_INPUT
    sToAdd : Str; // Text to append.
END_VAR

VAR
	_nNewLength	: INT;
END_VAR
Append := _this;

IF sToAdd = '' THEN
	RETURN;
END_IF

_nNewLength := Tc2_Standard.LEN(sToAdd) + _nLength;
IF _nNewLength > 255 THEN
	_nNewLength := 255;
END_IF

_sString := Tc2_Standard.CONCAT(_sString, sToAdd);
_nLength := _nNewLength;
END_METHOD

// Finds first match after position; outputs zero positions when not found.
METHOD FindFirstAfter : I_Strb
VAR_INPUT
    sToFind : Str;      // Text to find.
    nPosition : INT := 1; // One-based start position.
END_VAR
VAR_OUTPUT
    nStart : INT;       // Match start, or 0.
    nEnd : INT;         // Match end, or 0.
END_VAR

VAR
	_sTemp			: Str;
	_nOffset		: INT;
END_VAR
FindFirstAfter := _this;

IF sToFind = '' THEN
	RETURN;
END_IF

IF nPosition = 0 THEN
	RETURN;
END_IF

_sTemp := Tc2_Standard.MID(_sString, _nLength, nPosition);
IF (_nOffset := Tc2_Standard.FIND(_sTemp, sToFind)) <> 0 THEN
	nStart := nPosition + _nOffset - 1;
	nEnd := nPosition + _nOffset - 2 + Tc2_Standard.LEN(sToFind);
END_IF
END_METHOD

// Finds last match before position; outputs zero positions when not found.
METHOD FindLastBefore : I_Strb
VAR_INPUT
    sToFind : Str;        // Text to find.
    nPosition : INT := 256; // One-based end position; 256 means current length.
END_VAR
VAR_OUTPUT
    nStart : INT;         // Match start, or 0.
    nEnd : INT;           // Match end, or 0.
END_VAR
VAR
	_sTemp			: Str;
	_nFindLength	: INT := Tc2_Standard.LEN(sToFind);
	_nOffset		: INT;
END_VAR
FindLastBefore := _this;

IF sToFind = '' THEN
	RETURN;
END_IF

IF nPosition = 0 THEN
	RETURN;
END_IF

IF nPosition = 256 THEN
	nPosition := _nLength;
END_IF

REPEAT
	_sTemp := Tc2_Standard.MID(_sString, _nFindLength, nPosition);
	IF _sTemp = sToFind THEN
		nStart 	:= nPosition;
		nEnd	:= nPosition + _nFindLength - 1;
		RETURN;
	END_IF
UNTIL
	(nPosition := nPosition - 1) <= 0
END_REPEAT
END_METHOD

// Returns current text.
METHOD Get : Str
VAR_INPUT
END_VAR
Get := _sString;
END_METHOD

// Returns current length.
METHOD GetLength : INT
VAR_INPUT
END_VAR
GetLength := _nLength;
END_METHOD

// TRUE when text is found after position.
METHOD HasAfter : BOOL
VAR_INPUT
    sToFind : Str;      // Text to find.
    nPosition : INT := 0; // One-based start position.
END_VAR
VAR_OUTPUT
    nStart : INT;       // Match start, or 0.
    nEnd : INT;         // Match end, or 0.
END_VAR
FindFirstAfter(sToFind, nPosition, nStart => nStart, nEnd => nEnd);
HasAfter := nStart > 0;
END_METHOD

// TRUE when text is found before position.
METHOD HasBefore : BOOL
VAR_INPUT
    sToFind : Str;        // Text to find.
    nPosition : INT := 256; // One-based end position; 256 means current length.
END_VAR
VAR_OUTPUT
    nStart : INT;         // Match start, or 0.
    nEnd : INT;           // Match end, or 0.
END_VAR
IF nPosition = 256 THEN
	nPosition := Tc2_Standard.LEN(_sString);
END_IF

FindLastBefore(sToFind, nPosition, nStart => nStart, nEnd => nEnd);
HasBefore := nStart > 0;
END_METHOD

// Inserts text; no change when position is invalid.
METHOD Inject : I_Strb
VAR_INPUT
    nPosition : INT;    // One-based insert position.
    sToInject : Str;    // Text to insert.
END_VAR
VAR
	_nNewLength	: INT;
END_VAR
Inject := _this;

IF sToInject = '' THEN
	RETURN;
END_IF

IF nPosition = 0 THEN
	RETURN;
END_IF

IF nPosition > _nLength THEN
	RETURN;
END_IF

_nNewLength := Tc2_Standard.LEN(sToInject) + _nLength;
IF _nNewLength > 255 THEN
	_nNewLength := 255;
END_IF

_sString := Tc2_Standard.INSERT(_sString, sToInject, nPosition);
_nLength := _nNewLength;
END_METHOD

// TRUE when current length is 0.
METHOD IsEmpty : BOOL
VAR_INPUT
END_VAR
IsEmpty := _nLength = 0;
END_METHOD

// Outputs current length and returns this builder.
METHOD Length : I_Strb
VAR_OUTPUT
	nLen: INT; // Current length.
END_VAR
Length := _this;
nLen := _nLength;
END_METHOD

// Prepends text; truncates at 255 chars.
METHOD Prepend : I_Strb
VAR_INPUT
    sToAdd : Str; // Text to prepend.
END_VAR
VAR
	_nNewLength	: INT;
END_VAR
Prepend := _this;

IF sToAdd = '' THEN
	RETURN;
END_IF

_nNewLength := Tc2_Standard.LEN(sToAdd) + _nLength;
IF _nNewLength > 255 THEN
	_nNewLength := 255;
END_IF

_sString := Tc2_Standard.CONCAT(sToAdd, _sString);
_nLength := _nNewLength;
END_METHOD

// Removes text; no change when position or length is invalid.
METHOD Remove : I_Strb
VAR_INPUT
    nLength : INT;    // Characters to remove.
    nPosition : INT;  // One-based start position.
END_VAR

VAR
	_nPosition	: INT;
END_VAR
Remove := _this;

IF nPosition = 0 THEN
	RETURN;
END_IF

IF nPosition > _nLength THEN
	RETURN;
END_IF

IF nLength = 0 THEN
	RETURN;
END_IF

IF nLength + nPosition > _nLength THEN
	nLength := _nLength - nPosition + 1;
END_IF

_sString := Tc2_Standard.DELETE(_sString, nLength, nPosition);
_nLength := _nLength - nLength;
END_METHOD

// Sets current text.
METHOD Set : I_Strb
VAR_INPUT
    sValue : Str; // New text.
END_VAR
Set 		:= _this;

_sString 	:= sValue;
_nLength	:= Tc2_Standard.LEN(sValue);
END_METHOD

// Copies substring into sSlice; no change when position or length is invalid.
METHOD Slice : I_Strb
VAR_INPUT
    nLength : INT;   // Characters to copy.
    nPosition : INT; // One-based start position.
END_VAR
VAR_OUTPUT
    sSlice : Strb;   // Output slice builder.
END_VAR
Slice := _this;

IF nPosition = 0 THEN
	RETURN;
END_IF

IF nLength = 0 THEN
	RETURN;
END_IF

sSlice.Set(Tc2_Standard.MID(_sString, nLength, nPosition));
END_METHOD

// Splits text into left and right builders.
METHOD Split : I_Strb
VAR_INPUT
    nPosition : INT; // One-based split position.
END_VAR
VAR_OUTPUT
    sLeft : Strb;    // Left side.
    sRight : Strb;   // Right side.
END_VAR
Split := _this;

IF nPosition = 0 THEN
	RETURN;
END_IF

sLeft.Set(Tc2_Standard.LEFT(_sString, nPosition));
sRight.Set(Tc2_Standard.RIGHT(_sString, _nLength - nPosition));
END_METHOD

// Outputs current text and returns this builder.
METHOD Write : I_Strb;
VAR_OUTPUT
	sOut: Str; // Current text.
END_VAR
Write := _this;
sOut := _sString;
END_METHOD

END_FUNCTION_BLOCK

// ---- Utils/Strings/Strf/Strf.TcPOU
// String formatting helper namespace.
PROGRAM Strf

// Formats with one Tc2_Utilities argument.
METHOD Fmt : Str
VAR_INPUT
	sFormat			: Str; // Format string.
	tcArg			: Tc2_Utilities.T_Arg; // Format argument.
END_VAR
VAR
	_fmt			: Tc2_Utilities.FB_FormatString;
END_VAR
_fmt(sFormat := sFormat, arg1 := tcArg, sOut => Fmt);
END_METHOD

// Pads text; returns padded value.
METHOD Padding : Str
VAR_INPUT
    sValue       : Str;  // Text to pad.
    nLeftPadding : USINT := 0; // Minimum left-padded width.
    nRightPadding: USINT := 0; // Minimum right-padded width.
    sFillChar    : Ch := ' ';  // Fill character.
END_VAR
VAR
	_nLen		: INT := Tc2_Standard.LEN(sValue);
	_nLeftMiss	: INT;
	_nRightMiss	: INT;	

	i			: INT;
END_VAR
_nLeftMiss := nLeftPadding - _nLen;
_nRightMiss := nRightPadding - _nLen;

IF _nLeftMiss > 0 THEN
	FOR i := 1 TO _nleftMiss DO
		sValue := Tc2_Standard.CONCAT(sFillChar, sValue);
	END_FOR	
END_IF

IF _nRightMiss > 0 THEN
	FOR i := 1 TO _nRightMiss DO
		sValue := Tc2_Standard.CONCAT(sFillChar, sValue);
	END_FOR	
END_IF

Padding := sValue;
END_METHOD

// Formats TIME; returns empty string on invalid unit range.
METHOD SimpleTime : Str
VAR_INPUT
    tValue   : TIME;  // Time to format.
    sMinUnit : Str := 'MS'; // Minimum unit: MS, S, M, H, or D.
    sMaxUnit : Str := 'S';  // Maximum unit: MS, S, M, H, or D.
END_VAR
VAR
	_nMinUnit	: USINT;
	_nMaxUnit	: USINT;
	_sValues	: ARRAY[1..5] OF Strb;
	_nValues	: ARRAY[1..5] OF UINT;
	_sUnits   	: ARRAY[1..5] OF STRING := ['MS', 'S', 'M', 'H', 'D'];
	_stTime		: Tc2_Utilities.OTSTRUCT;
	_i			: USINT;
	_strb		: Strb;
END_VAR
FOR _i := 1 TO 5 DO
	IF _sUnits[_i] = sMinUnit THEN
		_nMinUnit := _i;
	END_IF
	IF _sUnits[_i] = sMaxUnit THEN
		_nMaxUnit := _i;
	END_IF
END_FOR

IF _nMaxUnit = 0 THEN
	RETURN;
END_IF

IF _nMinUnit = 0 THEN
	RETURN;
END_IF

IF _nMinUnit > _nMaxUnit THEN
	RETURN;
END_IF

_stTime := Tc2_Utilities.TIME_TO_OTSTRUCT(tValue);
_stTime.wDay := _stTime.wWeek * 7 + _stTime.wDay;

_nValues[1] := WORD_TO_UINT(_stTime.wMilliseconds);
_nValues[2] := WORD_TO_UINT(_stTime.wSecond);
_nValues[3] := WORD_TO_UINT(_stTime.wMinute);
_nValues[4] := WORD_TO_UINT(_stTime.wHour);
_nValues[5] := WORD_TO_UINT(_stTime.wDay);

_sValues[1].Set(Strf.Padding(UINT_TO_STRING(_nValues[1]), 3, 0, '0')).Append('ms');
_sValues[2].Set(Strf.Padding(UINT_TO_STRING(_nValues[2]), 2, 0, '0')).Append('s');
_sValues[3].Set(Strf.Padding(UINT_TO_STRING(_nValues[3]), 2, 0, '0')).Append('m');
_sValues[4].Set(Strf.Padding(UINT_TO_STRING(_nValues[4]), 2, 0, '0')).Append('h');
_sValues[5].Set(Strf.Padding(UINT_TO_STRING(_nValues[5]), 3, 0, '0')).Append('d');

IF _nMaxUnit < 5 THEN
    FOR _i := 5 TO _nMaxUnit + 1 BY -1 DO
        IF _nValues[_i] <> 0 THEN
            _strb.Append(_sValues[_i].Get()).Append(' ');
        END_IF
    END_FOR
END_IF

FOR _i := _nMaxUnit TO _nMinUnit BY -1 DO
    _strb.Append(_sValues[_i].Get()).Append(' ');
END_FOR

SimpleTime := _strb.Get();
END_METHOD

END_PROGRAM

// ---- Utils/Time/GetTaskCycleTime.TcPOU
// Returns current task cycle time in seconds.
FUNCTION GetTaskCycleTime : LREAL
VAR_IN_OUT CONSTANT
	taskInfo: ARRAY[*] OF PlcTaskSystemInfo; // Pass application _TaskInfo.
END_VAR

GetTaskCycleTime := UDINT_TO_LREAL(taskInfo[TC2_System.GETCURTASKINDEXEX()].CycleTime) / 10_000_000;

END_FUNCTION

// ---- Utils/Time/GetUnixTime.TcPOU
// Returns Unix-relative system time in 100 ns ticks.
FUNCTION GetUnixTime : ULINT
VAR_INPUT
	nOffset : LINT := 0; // Offset applied before epoch conversion.
END_VAR
VAR
END_VAR

GetUnixTime := Tc2_System.F_GetSystemTime() - LINT_TO_ULINT(11_644_473_678_000_000_0 + nOffset);

END_FUNCTION
